KUKA KRL program: MyProgram_289().src

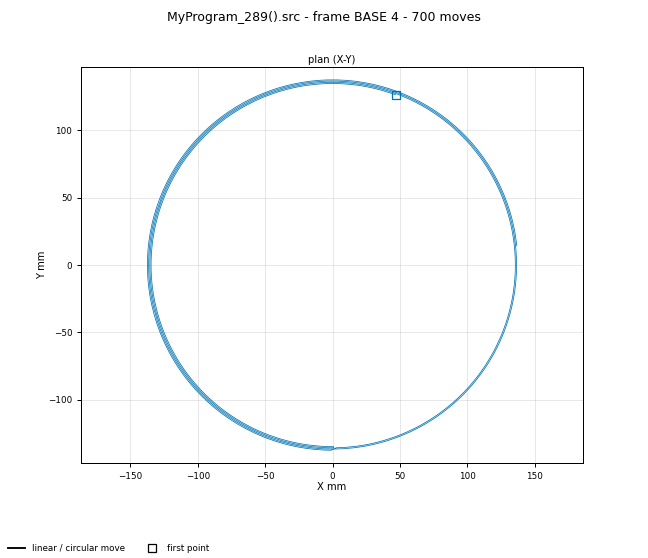
[picture p0: tool path of MyProgram_289().src in frame BASE 4, 700 of 700 moves have a stored position in this frame; points joined in program order, loops and branches not executed]
&ACCESS RVP
&REL 1
&PARAM TEMPLATE = C:\KRC\Roboter\Template\vorgabe
&PARAM EDITMASK = *
DEF MyProgram_289()
; ---- Setting reference (Base) ----
$BASE = BASE_DATA[4]

; --------------------------
; ---- Setting tool (TCP) ----
$TOOL = TOOL_DATA[3]
; --------------------------

$VEL.CP = VEL_APROX_PRINT
Startdeposition()
$VEL.CP = VEL_PRINT
LIN {X 46.739,Y 126.3738,Z 176,A 70.9873,B 7.2165,C 0.098,E1 7.2727,E2 380.9544} C_DIS
LIN {X 43.7934,Y 127.4239,Z 176,A 72.2694,B 7.2165,C 0.0975,E1 7.2693,E2 379.6782} C_DIS
LIN {X 36.8996,Y 129.5888,Z 176,A 75.2053,B 7.2165,C 0.0972,E1 7.2615,E2 376.7596} C_DIS
LIN {X 33.0824,Y 130.6146,Z 176,A 76.9284,B 7.2165,C 0.0952,E1 7.2569,E2 375.0317} C_DIS
LIN {X 29.3241,Y 131.5112,Z 176,A 78.6742,B 7.2166,C 0.0925,E1 7.2521,E2 373.2739} C_DIS
LIN {X 25.3274,Y 132.3373,Z 176,A 80.285,B 7.2166,C 0.0935,E1 7.2477,E2 371.6787} C_DIS
LIN {X 22.0563,Y 132.9217,Z 176,A 81.6963,B 7.2166,C 0.0929,E1 7.2438,E2 370.2679} C_DIS
LIN {X 18.536,Y 133.4592,Z 176,A 83.3203,B 7.2166,C 0.0905,E1 7.2393,E2 368.6313} C_DIS
LIN {X 13.6178,Y 134.0514,Z 176,A 85.4842,B 7.2166,C 0.089,E1 7.2333,E2 366.4611} C_DIS
LIN {X 9.065,Y 134.4361,Z 176,A 87.3794,B 7.2166,C 0.0893,E1 7.228,E2 364.5725} C_DIS
LIN {X 4.9514,Y 134.6487,Z 176,A 88.9717,B 7.2166,C 0.0915,E1 7.2236,E2 363.0001} C_DIS
LIN {X -0.1515,Y 134.74,Z 176,A 91.34,B 7.2166,C 0.0884,E1 7.2169,E2 360.6088} C_DIS
LIN {X -4.7786,Y 134.6554,Z 176,A 93.1801,B 7.2166,C 0.0905,E1 7.2118,E2 358.7852} C_DIS
LIN {X -8.4251,Y 134.4757,Z 176,A 94.6876,B 7.2166,C 0.0914,E1 7.2077,E2 357.2838} C_DIS
LIN {X -12.1995,Y 134.1876,Z 176,A 96.4009,B 7.2166,C 0.0902,E1 7.2029,E2 355.5589} C_DIS
LIN {X -16.1723,Y 133.7653,Z 176,A 97.9295,B 7.2166,C 0.0933,E1 7.1987,E2 354.0517} C_DIS
LIN {X -19.1655,Y 133.3692,Z 176,A 99.271,B 7.2166,C 0.0929,E1 7.1949,E2 352.7039} C_DIS
LIN {X -22.3244,Y 132.8769,Z 176,A 100.6251,B 7.2166,C 0.0936,E1 7.1912,E2 351.3514} C_DIS
LIN {X -25.9494,Y 132.2184,Z 176,A 102.3402,B 7.2166,C 0.0923,E1 7.1865,E2 349.6193} C_DIS
LIN {X -30.1027,Y 131.3334,Z 176,A 104.0357,B 7.2166,C 0.095,E1 7.1819,E2 347.9381} C_DIS
LIN {X -33.5303,Y 130.5009,Z 176,A 105.647,B 7.2166,C 0.0945,E1 7.1775,E2 346.3144} C_DIS
LIN {X -39.6195,Y 128.7825,Z 176,A 108.2833,B 7.2166,C 0.0974,E1 7.1704,E2 343.6864} C_DIS
LIN {X -42.7121,Y 127.79,Z 176,A 110.159,B 7.2166,C 0.0916,E1 7.1653,E2 341.7518} C_DIS
LIN {X -46.9366,Y 126.2998,Z 176,A 111.9973,B 7.2166,C 0.0944,E1 7.1605,E2 339.923} C_DIS
LIN {X -50.7015,Y 124.8361,Z 176,A 113.2648,B 7.2165,C 0.1026,E1 7.1574,E2 338.7113} C_DIS
LIN {X -53.8637,Y 123.5048,Z 176,A 114.743,B 7.2165,C 0.104,E1 7.1536,E2 337.2318} C_DIS
LIN {X -56.9194,Y 122.1266,Z 176,A 116.2037,B 7.2165,C 0.1052,E1 7.1499,E2 335.7679} C_DIS
LIN {X -63.2599,Y 118.9673,Z 176,A 119.0396,B 7.2163,C 0.1116,E1 7.1429,E2 332.9558} C_DIS
LIN {X -65.7728,Y 117.5973,Z 176,A 120.5687,B 7.2163,C 0.109,E1 7.139,E2 331.3901} C_DIS
LIN {X -70.8593,Y 114.6044,Z 176,A 122.972,B 7.2163,C 0.1142,E1 7.1333,E2 329.0017} C_DIS
LIN {X -73.968,Y 112.6226,Z 176,A 124.66,B 7.2163,C 0.115,E1 7.1293,E2 327.3004} C_DIS
LIN {X -78.7898,Y 109.3041,Z 176,A 127.0345,B 7.2163,C 0.1206,E1 7.1239,E2 324.9419} C_DIS
LIN {X -81.5123,Y 107.2894,Z 176,A 128.6056,B 7.2162,C 0.1214,E1 7.1204,E2 323.3563} C_DIS
LIN {X -84.8943,Y 104.6336,Z 176,A 130.4274,B 7.2162,C 0.1248,E1 7.1164,E2 321.5369} C_DIS
LIN {X -87.9949,Y 102.0392,Z 176,A 132.5845,B 7.2162,C 0.1222,E1 7.1117,E2 319.3282} C_DIS
LIN {X -90.9601,Y 99.4054,Z 176,A 133.9926,B 7.2161,C 0.1291,E1 7.1089,E2 317.9555} C_DIS
LIN {X -95.2089,Y 95.344,Z 176,A 136.3018,B 7.2159,C 0.1366,E1 7.1043,E2 315.6716} C_DIS
LIN {X -97.6628,Y 92.8289,Z 176,A 138.2509,B 7.2159,C 0.1338,E1 7.1004,E2 313.6688} C_DIS
LIN {X -99.9947,Y 90.3119,Z 176,A 139.2657,B 7.2158,C 0.1427,E1 7.0986,E2 312.7091} C_DIS
LIN {X -102.1705,Y 87.8423,Z 176,A 141.0418,B 7.2158,C 0.1409,E1 7.0953,E2 310.8887} C_DIS
LIN {X -105.7645,Y 83.4809,Z 176,A 143.5332,B 7.2158,C 0.1452,E1 7.0909,E2 308.3889} C_DIS
LIN {X -108.9535,Y 79.2734,Z 176,A 145.5935,B 7.2156,C 0.1527,E1 7.0875,E2 306.3532} C_DIS
LIN {X -112.011,Y 74.8908,Z 176,A 147.5992,B 7.2154,C 0.1615,E1 7.0844,E2 304.3819} C_DIS
LIN {X -113.5489,Y 72.538,Z 176,A 149.4424,B 7.2155,C 0.1562,E1 7.0815,E2 302.4612} C_DIS
LIN {X -115.46,Y 69.4557,Z 176,A 150.6583,B 7.2153,C 0.1642,E1 7.0798,E2 301.2866} C_DIS
LIN {X -117.0516,Y 66.7384,Z 176,A 152.5358,B 7.2154,C 0.1607,E1 7.0771,E2 299.3447} C_DIS
LIN {X -119.1423,Y 62.9266,Z 176,A 153.6832,B 7.2151,C 0.1743,E1 7.0757,E2 298.2845} C_DIS
LIN {X -120.2429,Y 60.7975,Z 176,A 154.9377,B 7.2151,C 0.1739,E1 7.0741,E2 297.0024} C_DIS
LIN {X -121.7624,Y 57.6944,Z 176,A 156.459,B 7.2151,C 0.1771,E1 7.0722,E2 295.4761} C_DIS
LIN {X -123.8033,Y 53.1733,Z 176,A 158.5577,B 7.2149,C 0.1828,E1 7.0699,E2 293.3808} C_DIS
LIN {X -125.0493,Y 50.1725,Z 176,A 160.0003,B 7.2149,C 0.1857,E1 7.0683,E2 291.9321} C_DIS
LIN {X -127.412,Y 43.8276,Z 176,A 162.9337,B 7.2146,C 0.1929,E1 7.0655,E2 288.9949} C_DIS
LIN {X -128.6112,Y 40.1791,Z 176,A 164.7288,B 7.2146,C 0.1954,E1 7.064,E2 287.1816} C_DIS
LIN {X -129.7986,Y 36.1515,Z 176,A 166.3975,B 7.2144,C 0.2018,E1 7.0627,E2 285.5288} C_DIS
LIN {X -130.7393,Y 32.5908,Z 176,A 167.9676,B 7.2143,C 0.2061,E1 7.0616,E2 283.9597} C_DIS
LIN {X -131.4143,Y 29.7485,Z 176,A 169.2369,B 7.2142,C 0.2092,E1 7.0608,E2 282.6882} C_DIS
LIN {X -132.1055,Y 26.5122,Z 176,A 170.6847,B 7.2141,C 0.2127,E1 7.06,E2 281.2367} C_DIS
LIN {X -132.7822,Y 22.8924,Z 176,A 172.4282,B 7.2141,C 0.215,E1 7.0591,E2 279.473} C_DIS
LIN {X -133.3823,Y 19.0741,Z 176,A 173.9886,B 7.2138,C 0.2207,E1 7.0585,E2 277.9242} C_DIS
LIN {X -133.8523,Y 15.4428,Z 176,A 175.6627,B 7.2138,C 0.2237,E1 7.0579,E2 276.2371} C_DIS
LIN {X -134.2767,Y 11.1572,Z 176,A 177.4463,B 7.2136,C 0.2295,E1 7.0575,E2 274.461} C_DIS
LIN {X -134.5431,Y 7.2873,Z 176,A 179.2247,B 7.2135,C 0.2327,E1 7.0572,E2 272.6683} C_DIS
LIN {X -134.7031,Y 3.1775,Z 176,A -178.9548,B 7.2133,C 0.2368,E1 7.057,E2 270.8405} C_DIS
LIN {X -134.7368,Y -0.9717,Z 176,A -177.1983,B 7.2132,C 0.242,E1 7.057,E2 269.0864} C_DIS
LIN {X -134.6421,Y -5.1206,Z 176,A -175.4593,B 7.213,C 0.2474,E1 7.0572,E2 267.352} C_DIS
LIN {X -134.429,Y -9.1625,Z 176,A -173.6351,B 7.2129,C 0.251,E1 7.0575,E2 265.5166} C_DIS
LIN {X -134.1144,Y -12.9613,Z 176,A -172.077,B 7.2127,C 0.2564,E1 7.0579,E2 263.9675} C_DIS
LIN {X -133.7153,Y -16.5917,Z 176,A -170.4743,B 7.2125,C 0.2602,E1 7.0584,E2 262.36} C_DIS
LIN {X -133.1806,Y -20.4353,Z 176,A -168.761,B 7.2124,C 0.2641,E1 7.0591,E2 260.6401} C_DIS
LIN {X -132.5589,Y -24.1444,Z 176,A -167.1691,B 7.2122,C 0.2687,E1 7.0599,E2 259.0503} C_DIS
LIN {X -131.7289,Y -28.322,Z 176,A -165.3319,B 7.212,C 0.2735,E1 7.0609,E2 257.2112} C_DIS
LIN {X -130.0027,Y -35.4179,Z 176,A -161.457,B 7.212,C 0.2724,E1 7.0637,E2 253.2431} C_DIS
LIN {X -128.5121,Y -40.4909,Z 176,A -159.9882,B 7.2115,C 0.2884,E1 7.0648,E2 251.8727} C_DIS
LIN {X -127.1443,Y -44.5999,Z 176,A -157.774,B 7.2115,C 0.2886,E1 7.0668,E2 249.6135} C_DIS
LIN {X -125.5592,Y -48.882,Z 176,A -155.9827,B 7.2112,C 0.2957,E1 7.0686,E2 247.8421} C_DIS
LIN {X -124.2324,Y -52.1626,Z 176,A -154.4732,B 7.211,C 0.2996,E1 7.0702,E2 246.333} C_DIS
LIN {X -122.9434,Y -55.1316,Z 176,A -153.0961,B 7.2109,C 0.3031,E1 7.0717,E2 244.9566} C_DIS
LIN {X -121.2485,Y -58.7688,Z 176,A -151.3637,B 7.2107,C 0.3072,E1 7.0738,E2 243.2219} C_DIS
LIN {X -120.0628,Y -61.1512,Z 176,A -149.7902,B 7.2108,C 0.3043,E1 7.0759,E2 241.5939} C_DIS
LIN {X -118.2615,Y -64.5696,Z 176,A -148.0643,B 7.2107,C 0.3073,E1 7.0782,E2 239.8586} C_DIS
LIN {X -116.2697,Y -68.0917,Z 176,A -147.0058,B 7.2101,C 0.3201,E1 7.0796,E2 238.8836} C_DIS
LIN {X -114.7894,Y -70.5584,Z 176,A -145.4501,B 7.2101,C 0.3188,E1 7.0819,E2 237.2872} C_DIS
LIN {X -112.3758,Y -74.3429,Z 176,A -143.133,B 7.2102,C 0.3179,E1 7.0855,E2 234.9198} C_DIS
LIN {X -110.1367,Y -77.6209,Z 176,A -141.8141,B 7.2098,C 0.3267,E1 7.0875,E2 233.6479} C_DIS
LIN {X -108.2709,Y -80.2035,Z 176,A -139.8806,B 7.2101,C 0.3221,E1 7.0909,E2 231.6424} C_DIS
LIN {X -105.3441,Y -84.0103,Z 176,A -138.3443,B 7.2095,C 0.3333,E1 7.0934,E2 230.1703} C_DIS
LIN {X -102.7193,Y -87.2,Z 176,A -136.5236,B 7.2095,C 0.3362,E1 7.0967,E2 228.3423} C_DIS
LIN {X -99.0727,Y -91.322,Z 176,A -134.4345,B 7.209,C 0.3444,E1 7.1005,E2 226.2854} C_DIS
LIN {X -97.1061,Y -93.4113,Z 176,A -132.8728,B 7.2091,C 0.3423,E1 7.1036,E2 224.6813} C_DIS
LIN {X -93.9427,Y -96.5917,Z 176,A -130.9489,B 7.209,C 0.3457,E1 7.1074,E2 222.7558} C_DIS
LIN {X -90.755,Y -99.5926,Z 176,A -129.0641,B 7.2088,C 0.3489,E1 7.1113,E2 220.8685} C_DIS
LIN {X -87.4295,Y -102.5242,Z 176,A -127.1743,B 7.2086,C 0.3522,E1 7.1153,E2 218.9786} C_DIS
LIN {X -83.2923,Y -105.9126,Z 176,A -125.0607,B 7.2083,C 0.3584,E1 7.1199,E2 216.8855} C_DIS
LIN {X -80.0894,Y -108.3546,Z 176,A -122.7965,B 7.2086,C 0.3535,E1 7.1251,E2 214.5521} C_DIS
LIN {X -76.7889,Y -110.7185,Z 176,A -121.6345,B 7.2081,C 0.3641,E1 7.1276,E2 213.4614} C_DIS
LIN {X -73.9442,Y -112.6382,Z 176,A -119.9283,B 7.2081,C 0.3628,E1 7.1316,E2 211.7243} C_DIS
LIN {X -70.1568,Y -115.0358,Z 176,A -117.9951,B 7.2081,C 0.3651,E1 7.1362,E2 209.7879} C_DIS
LIN {X -66.356,Y -117.2694,Z 176,A -116.0672,B 7.2079,C 0.3669,E1 7.1409,E2 207.8532} C_DIS
LIN {X -62.4442,Y -119.3956,Z 176,A -114.285,B 7.2077,C 0.3708,E1 7.1452,E2 206.0849} C_DIS
LIN {X -59.2266,Y -121.0245,Z 176,A -112.754,B 7.2077,C 0.3727,E1 7.1491,E2 204.5543} C_DIS
LIN {X -55.9568,Y -122.5717,Z 176,A -111.1959,B 7.2076,C 0.3741,E1 7.153,E2 202.9936} C_DIS
LIN {X -51.5409,Y -124.492,Z 176,A -109.084,B 7.2075,C 0.3753,E1 7.1585,E2 200.8733} C_DIS
LIN {X -46.8002,Y -126.3509,Z 176,A -106.8561,B 7.2075,C 0.3763,E1 7.1643,E2 198.6373} C_DIS
LIN {X -40.0759,Y -128.6423,Z 176,A -103.9389,B 7.2072,C 0.3803,E1 7.172,E2 195.7328} C_DIS
LIN {X -37.4879,Y -129.4195,Z 176,A -102.7989,B 7.2072,C 0.3812,E1 7.175,E2 194.5936} C_DIS
LIN {X -34.6618,Y -130.2043,Z 176,A -101.5236,B 7.2072,C 0.3816,E1 7.1785,E2 193.3145} C_DIS
LIN {X -31.4986,Y -131.0055,Z 176,A -100.1131,B 7.2072,C 0.382,E1 7.1823,E2 191.9007} C_DIS
LIN {X -28.3558,Y -131.7216,Z 176,A -98.766,B 7.2071,C 0.3831,E1 7.186,E2 190.5562} C_DIS
LIN {X -25.1394,Y -132.3732,Z 176,A -97.3637,B 7.2071,C 0.3836,E1 7.1898,E2 189.1526} C_DIS
LIN {X -22.007,Y -132.9299,Z 176,A -95.9846,B 7.2071,C 0.3836,E1 7.1936,E2 187.7698} C_DIS
LIN {X -18.2836,Y -133.4951,Z 176,A -93.8301,B 7.2075,C 0.3755,E1 7.1998,E2 185.5446} C_DIS
LIN {X -13.7352,Y -134.0391,Z 176,A -92.4659,B 7.207,C 0.3851,E1 7.2034,E2 184.2538} C_DIS
LIN {X -10.8566,Y -134.3021,Z 176,A -91.1132,B 7.207,C 0.3833,E1 7.2072,E2 182.885} C_DIS
LIN {X -6.8342,Y -134.5659,Z 176,A -89.1612,B 7.2073,C 0.3795,E1 7.2127,E2 180.902} C_DIS
LIN {X -3.396,Y -134.697,Z 176,A -87.6016,B 7.2073,C 0.3779,E1 7.2171,E2 179.3295} C_DIS
LIN {X 0.5077,Y -134.7387,Z 176,A -86.3072,B 7.2071,C 0.3836,E1 7.2206,E2 178.0808} C_DIS
LIN {X 0.5077,Y -134.7387,Z 176,A -86.3072,B 7.2071,C 0.3836,E1 7.2206,E2 178.0808} C_DIS
Enddeposition()
LIN {X 0.996,Y -135.641,Z 176,A -86.1239,B 7.1241,C 0.3885,E1 7.1383,E2 177.9572} C_DIS
Startdeposition()
$VEL.CP = VEL_PRINT
LIN {X -4.7077,Y -135.5642,Z 176,A -89.0853,B 7.1236,C 0.3974,E1 7.1299,E2 180.9899} C_DIS
LIN {X -9.5873,Y -135.3061,Z 176,A -91.2415,B 7.1236,C 0.3987,E1 7.1238,E2 183.1586} C_DIS
LIN {X -13.0181,Y -135.0188,Z 176,A -93.0667,B 7.1232,C 0.4042,E1 7.1186,E2 185.0311} C_DIS
LIN {X -16.8806,Y -134.5909,Z 176,A -94.558,B 7.1234,C 0.4015,E1 7.1145,E2 186.5041} C_DIS
LIN {X -22.3201,Y -133.7959,Z 176,A -96.6569,B 7.1236,C 0.3974,E1 7.1088,E2 188.5757} C_DIS
LIN {X -26.2786,Y -133.0773,Z 176,A -98.4709,B 7.1236,C 0.3984,E1 7.1038,E2 190.4048} C_DIS
LIN {X -30.3133,Y -132.2143,Z 176,A -100.0712,B 7.1236,C 0.3954,E1 7.0995,E2 191.9875} C_DIS
LIN {X -33.4857,Y -131.4466,Z 176,A -101.4995,B 7.1236,C 0.3954,E1 7.0956,E2 193.4224} C_DIS
LIN {X -36.965,Y -130.5116,Z 176,A -103.0564,B 7.1237,C 0.3949,E1 7.0914,E2 194.9841} C_DIS
LIN {X -43.7768,Y -128.3882,Z 176,A -105.9689,B 7.1239,C 0.3911,E1 7.0837,E2 197.8845} C_DIS
LIN {X -47.6211,Y -127.0106,Z 176,A -107.8293,B 7.1239,C 0.3916,E1 7.0787,E2 199.7621} C_DIS
LIN {X -51.2699,Y -125.5835,Z 176,A -109.6042,B 7.1239,C 0.3917,E1 7.0741,E2 201.5524} C_DIS
LIN {X -54.6493,Y -124.1513,Z 176,A -110.9764,B 7.1241,C 0.3876,E1 7.0706,E2 202.9023} C_DIS
LIN {X -57.1447,Y -123.0202,Z 176,A -112.1786,B 7.1241,C 0.3869,E1 7.0676,E2 204.1103} C_DIS
LIN {X -60.2043,Y -121.5521,Z 176,A -113.6365,B 7.1242,C 0.3856,E1 7.0639,E2 205.5713} C_DIS
LIN {X -63.7521,Y -119.7318,Z 176,A -115.3454,B 7.1243,C 0.3839,E1 7.0597,E2 207.2833} C_DIS
LIN {X -67.5396,Y -117.6373,Z 176,A -117.2786,B 7.1243,C 0.383,E1 7.0549,E2 209.2297} C_DIS
LIN {X -71.4568,Y -115.2995,Z 176,A -119.2047,B 7.1245,C 0.3803,E1 7.0503,E2 211.1557} C_DIS
LIN {X -75.2415,Y -112.8659,Z 176,A -121.1047,B 7.1247,C 0.3775,E1 7.0459,E2 213.0554} C_DIS
LIN {X -80.6564,Y -109.0628,Z 176,A -123.9768,B 7.1248,C 0.3741,E1 7.0393,E2 215.9369} C_DIS
LIN {X -84.2255,Y -106.3303,Z 176,A -125.9951,B 7.1249,C 0.3725,E1 7.0349,E2 217.9698} C_DIS
LIN {X -87.0011,Y -104.0714,Z 176,A -127.4206,B 7.1251,C 0.3687,E1 7.0318,E2 219.3843} C_DIS
LIN {X -90.5428,Y -101.0048,Z 176,A -129.3934,B 7.1253,C 0.3651,E1 7.0277,E2 221.356} C_DIS
LIN {X -93.9342,Y -97.8593,Z 176,A -131.3841,B 7.1255,C 0.3618,E1 7.0236,E2 223.3508} C_DIS
LIN {X -97.1434,Y -94.6747,Z 176,A -133.3331,B 7.1256,C 0.3586,E1 7.0198,E2 225.3042} C_DIS
LIN {X -100.7337,Y -90.8447,Z 176,A -135.4229,B 7.1259,C 0.3524,E1 7.0159,E2 227.3774} C_DIS
LIN {X -102.6613,Y -88.6604,Z 176,A -136.8314,B 7.1259,C 0.3522,E1 7.0132,E2 228.8076} C_DIS
LIN {X -105.5562,Y -85.1931,Z 176,A -138.734,B 7.1262,C 0.348,E1 7.0099,E2 230.7089} C_DIS
LIN {X -110.1768,Y -79.1273,Z 176,A -141.7148,B 7.1266,C 0.3377,E1 7.0049,E2 233.6586} C_DIS
LIN {X -113.3344,Y -74.5338,Z 176,A -144.1448,B 7.1269,C 0.3332,E1 7.0011,E2 236.0971} C_DIS
LIN {X -114.9573,Y -72.0066,Z 176,A -145.7504,B 7.1268,C 0.3345,E1 6.9986,E2 237.744} C_DIS
LIN {X -117.317,Y -68.0936,Z 176,A -148.2444,B 7.1267,C 0.3369,E1 6.995,E2 240.3066} C_DIS
LIN {X -119.8043,Y -63.614,Z 176,A -149.6976,B 7.1273,C 0.3226,E1 6.9932,E2 241.671} C_DIS
LIN {X -121.1064,Y -61.0976,Z 176,A -151.0675,B 7.1273,C 0.3218,E1 6.9914,E2 243.0616} C_DIS
LIN {X -123.2128,Y -56.7282,Z 176,A -153.0883,B 7.1276,C 0.3162,E1 6.989,E2 245.0778} C_DIS
LIN {X -124.5702,Y -53.6818,Z 176,A -154.5239,B 7.1278,C 0.3129,E1 6.9874,E2 246.5159} C_DIS
LIN {X -125.973,Y -50.3035,Z 176,A -156.101,B 7.1279,C 0.3092,E1 6.9857,E2 248.096} C_DIS
LIN {X -127.2111,Y -47.0857,Z 176,A -157.6421,B 7.1281,C 0.3064,E1 6.9842,E2 249.6467} C_DIS
LIN {X -128.4332,Y -43.6467,Z 176,A -159.1463,B 7.1282,C 0.3018,E1 6.9828,E2 251.1454} C_DIS
LIN {X -129.8934,Y -39.0844,Z 176,A -161.797,B 7.1282,C 0.304,E1 6.9806,E2 253.8717} C_DIS
LIN {X -131.1515,Y -34.6251,Z 176,A -163.5893,B 7.1285,C 0.2966,E1 6.9793,E2 255.6424} C_DIS
LIN {X -132.063,Y -30.9751,Z 176,A -164.8088,B 7.1288,C 0.2876,E1 6.9785,E2 256.8155} C_DIS
LIN {X -132.9914,Y -26.7009,Z 176,A -166.6352,B 7.129,C 0.2822,E1 6.9775,E2 258.6379} C_DIS
LIN {X -133.5606,Y -23.6881,Z 176,A -168.0202,B 7.1291,C 0.2797,E1 6.9768,E2 260.0329} C_DIS
LIN {X -134.1555,Y -20.0583,Z 176,A -169.789,B 7.1292,C 0.2779,E1 6.976,E2 261.827} C_DIS
LIN {X -134.6974,Y -16.0048,Z 176,A -171.411,B 7.1295,C 0.2717,E1 6.9754,E2 263.4348} C_DIS
LIN {X -135.117,Y -11.9696,Z 176,A -173.227,B 7.1295,C 0.2681,E1 6.9749,E2 265.262} C_DIS
LIN {X -135.4001,Y -8.1499,Z 176,A -174.7919,B 7.1298,C 0.2628,E1 6.9746,E2 266.8191} C_DIS
LIN {X -135.5792,Y -4.2544,Z 176,A -176.5543,B 7.1299,C 0.2595,E1 6.9745,E2 268.5943} C_DIS
LIN {X -135.6467,Y -0.306,Z 176,A -178.188,B 7.1301,C 0.2543,E1 6.9745,E2 270.2224} C_DIS
LIN {X -135.5959,Y 3.6532,Z 176,A -179.9351,B 7.1302,C 0.2504,E1 6.9745,E2 271.9772} C_DIS
LIN {X -135.4109,Y 7.9751,Z 176,A 178.1962,B 7.1304,C 0.2456,E1 6.9748,E2 273.8494} C_DIS
LIN {X -135.1544,Y 11.5263,Z 176,A 176.6976,B 7.1305,C 0.2412,E1 6.9751,E2 275.3459} C_DIS
LIN {X -134.7366,Y 15.6763,Z 176,A 174.8477,B 7.1307,C 0.2373,E1 6.9756,E2 277.205} C_DIS
LIN {X -134.27,Y 19.264,Z 176,A 173.3565,B 7.1308,C 0.2325,E1 6.9762,E2 278.6904} C_DIS
LIN {X -133.7599,Y 22.5356,Z 176,A 171.8778,B 7.1309,C 0.2294,E1 6.9769,E2 280.1776} C_DIS
LIN {X -132.9543,Y 26.8828,Z 176,A 170.0024,B 7.1311,C 0.2243,E1 6.9779,E2 282.0523} C_DIS
LIN {X -132.2009,Y 30.3717,Z 176,A 168.4755,B 7.1312,C 0.2203,E1 6.9788,E2 283.5801} C_DIS
LIN {X -131.3092,Y 34.0272,Z 176,A 166.6861,B 7.1312,C 0.2182,E1 6.98,E2 285.3924} C_DIS
LIN {X -130.1443,Y 38.2357,Z 176,A 164.9617,B 7.1315,C 0.2117,E1 6.9813,E2 287.1004} C_DIS
LIN {X -128.9768,Y 42.0127,Z 176,A 162.8066,B 7.1315,C 0.2129,E1 6.9832,E2 289.3128} C_DIS
LIN {X -127.6927,Y 45.7614,Z 176,A 161.1611,B 7.1315,C 0.208,E1 6.9848,E2 290.9532} C_DIS
LIN {X -126.3735,Y 49.2871,Z 176,A 159.9412,B 7.1318,C 0.1993,E1 6.9859,E2 292.1268} C_DIS
LIN {X -125.0343,Y 52.5927,Z 176,A 158.3786,B 7.1319,C 0.196,E1 6.9876,E2 293.6948} C_DIS
LIN {X -123.749,Y 55.5487,Z 176,A 156.9618,B 7.132,C 0.193,E1 6.9892,E2 295.1171} C_DIS
LIN {X -121.9613,Y 59.3748,Z 176,A 155.0967,B 7.132,C 0.1894,E1 6.9915,E2 296.9904} C_DIS
LIN {X -120.2137,Y 62.8344,Z 176,A 152.9644,B 7.132,C 0.1912,E1 6.9943,E2 299.1805} C_DIS
LIN {X -117.9396,Y 67.0095,Z 176,A 151.4736,B 7.1323,C 0.1799,E1 6.9962,E2 300.6073} C_DIS
LIN {X -114.947,Y 72.0231,Z 176,A 149.1216,B 7.1325,C 0.1724,E1 6.9996,E2 302.9432} C_DIS
LIN {X -113.2159,Y 74.7139,Z 176,A 147.4934,B 7.1325,C 0.1725,E1 7.0021,E2 304.6036} C_DIS
LIN {X -110.5111,Y 78.6598,Z 176,A 145.412,B 7.1326,C 0.1685,E1 7.0055,E2 306.6903} C_DIS
LIN {X -107.3939,Y 82.8645,Z 176,A 143.3778,B 7.1328,C 0.1612,E1 7.0088,E2 308.7012} C_DIS
LIN {X -105.7022,Y 85.0121,Z 176,A 142.0358,B 7.1328,C 0.1609,E1 7.0112,E2 310.0647} C_DIS
LIN {X -102.2429,Y 89.1424,Z 176,A 139.7364,B 7.1328,C 0.1562,E1 7.0154,E2 312.3649} C_DIS
LIN {X -98.349,Y 93.4217,Z 176,A 137.3126,B 7.133,C 0.1508,E1 7.02,E2 314.784} C_DIS
LIN {X -95.5885,Y 96.2435,Z 176,A 135.0858,B 7.133,C 0.1545,E1 7.0245,E2 317.0763} C_DIS
LIN {X -92.2942,Y 99.4072,Z 176,A 133.0505,B 7.133,C 0.1521,E1 7.0287,E2 319.1225} C_DIS
LIN {X -88.5973,Y 102.7157,Z 176,A 131.6203,B 7.1332,C 0.1396,E1 7.0315,E2 320.4713} C_DIS
LIN {X -85.7718,Y 105.0866,Z 176,A 129.8866,B 7.1332,C 0.139,E1 7.0353,E2 322.2247} C_DIS
LIN {X -82.7111,Y 107.5128,Z 176,A 128.1632,B 7.1332,C 0.137,E1 7.0391,E2 323.9556} C_DIS
LIN {X -78.4225,Y 110.6788,Z 176,A 125.9224,B 7.1334,C 0.1331,E1 7.0441,E2 326.1931} C_DIS
LIN {X -75.3263,Y 112.8093,Z 176,A 124.3183,B 7.1334,C 0.1307,E1 7.0479,E2 327.7979} C_DIS
LIN {X -71.4969,Y 115.2745,Z 176,A 121.5698,B 7.1333,C 0.1387,E1 7.0546,E2 330.643} C_DIS
LIN {X -65.9584,Y 118.5308,Z 176,A 119.6722,B 7.1335,C 0.124,E1 7.059,E2 332.4413} C_DIS
LIN {X -58.2367,Y 122.5071,Z 176,A 116.0304,B 7.1336,C 0.1189,E1 7.068,E2 336.0772} C_DIS
LIN {X -55.0069,Y 123.9913,Z 176,A 114.4758,B 7.1336,C 0.1178,E1 7.072,E2 337.637} C_DIS
LIN {X -51.4984,Y 125.4913,Z 176,A 111.9759,B 7.1335,C 0.1282,E1 7.0788,E2 340.2415} C_DIS
LIN {X -45.5058,Y 127.7848,Z 176,A 110.1969,B 7.1337,C 0.1127,E1 7.0831,E2 341.9077} C_DIS
LIN {X -42.6383,Y 128.7691,Z 176,A 108.8279,B 7.1337,C 0.1127,E1 7.0868,E2 343.2864} C_DIS
LIN {X -39.2995,Y 129.8276,Z 176,A 106.9759,B 7.1337,C 0.1168,E1 7.0918,E2 345.182} C_DIS
LIN {X -35.5706,Y 130.8993,Z 176,A 105.8086,B 7.1337,C 0.1089,E1 7.0948,E2 346.2919} C_DIS
LIN {X -32.1245,Y 131.7863,Z 176,A 104.1734,B 7.1337,C 0.1097,E1 7.0993,E2 347.942} C_DIS
LIN {X -28.5733,Y 132.6012,Z 176,A 102.6646,B 7.1337,C 0.1083,E1 7.1034,E2 349.4462} C_DIS
LIN {X -24.9362,Y 133.3342,Z 176,A 101.138,B 7.1338,C 0.1069,E1 7.1075,E2 350.967} C_DIS
LIN {X -21.8816,Y 133.869,Z 176,A 99.7491,B 7.1338,C 0.1074,E1 7.1114,E2 352.3647} C_DIS
LIN {X -17.8333,Y 134.4677,Z 176,A 98.0158,B 7.1338,C 0.1068,E1 7.1162,E2 354.0976} C_DIS
LIN {X -14.0847,Y 134.9124,Z 176,A 96.3394,B 7.1338,C 0.1075,E1 7.1209,E2 355.7829} C_DIS
LIN {X -9.9702,Y 135.2781,Z 176,A 94.6732,B 7.1338,C 0.106,E1 7.1255,E2 357.4388} C_DIS
LIN {X -6.0142,Y 135.5136,Z 176,A 92.8868,B 7.1338,C 0.1074,E1 7.1305,E2 359.2379} C_DIS
LIN {X -1.7426,Y 135.6343,Z 176,A 91.0375,B 7.1338,C 0.108,E1 7.1357,E2 361.0916} C_DIS
LIN {X 3.4099,Y 135.6027,Z 176,A 89.0337,B 7.1338,C 0.1055,E1 7.1412,E2 363.0737} C_DIS
LIN {X 6.5509,Y 135.487,Z 176,A 87.6793,B 7.1338,C 0.106,E1 7.145,E2 364.4308} C_DIS
LIN {X 10.1232,Y 135.267,Z 176,A 86.132,B 7.1338,C 0.1069,E1 7.1493,E2 365.9817} C_DIS
LIN {X 14.2563,Y 134.8939,Z 176,A 84.4263,B 7.1338,C 0.1067,E1 7.154,E2 367.6812} C_DIS
LIN {X 18.3399,Y 134.4013,Z 176,A 82.5974,B 7.1338,C 0.1087,E1 7.1591,E2 369.5205} C_DIS
LIN {X 22.296,Y 133.7999,Z 176,A 81.0367,B 7.1338,C 0.1075,E1 7.1634,E2 371.0651} C_DIS
LIN {X 25.7585,Y 133.177,Z 176,A 79.565,B 7.1338,C 0.1081,E1 7.1674,E2 372.5347} C_DIS
LIN {X 28.7296,Y 132.5674,Z 176,A 78.3064,B 7.1338,C 0.1085,E1 7.1709,E2 373.7902} C_DIS
LIN {X 31.9423,Y 131.8302,Z 176,A 76.8821,B 7.1338,C 0.1099,E1 7.1747,E2 375.218} C_DIS
LIN {X 35.7578,Y 130.8492,Z 176,A 74.5988,B 7.1336,C 0.1209,E1 7.1811,E2 377.5752} C_DIS
LIN {X 40.665,Y 129.4073,Z 176,A 73.1781,B 7.1337,C 0.111,E1 7.1847,E2 378.9069} C_DIS
LIN {X 45.3873,Y 127.8276,Z 176,A 71.001,B 7.1337,C 0.1141,E1 7.1904,E2 381.0925} C_DIS
LIN {X 48.392,Y 126.7214,Z 176,A 69.4815,B 7.1337,C 0.1182,E1 7.1945,E2 382.6319} C_DIS
LIN {X 52.4009,Y 125.1144,Z 176,A 67.8358,B 7.1337,C 0.1173,E1 7.1986,E2 384.2559} C_DIS
LIN {X 55.5295,Y 123.7576,Z 176,A 66.4224,B 7.1337,C 0.1185,E1 7.2023,E2 385.666} C_DIS
LIN {X 58.659,Y 122.3054,Z 176,A 64.9734,B 7.1336,C 0.1202,E1 7.2059,E2 387.1138} C_DIS
LIN {X 61.9204,Y 120.6875,Z 176,A 63.4073,B 7.1336,C 0.1226,E1 7.2098,E2 388.6834} C_DIS
LIN {X 66.0072,Y 118.5038,Z 176,A 61.4124,B 7.1335,C 0.126,E1 7.2147,E2 390.6829} C_DIS
LIN {X 69.864,Y 116.2719,Z 176,A 59.5271,B 7.1335,C 0.1288,E1 7.2193,E2 392.5686} C_DIS
LIN {X 73.7625,Y 113.838,Z 176,A 57.4366,B 7.1333,C 0.1342,E1 7.2242,E2 394.6773} C_DIS
LIN {X 76.5449,Y 111.9863,Z 176,A 56.522,B 7.1335,C 0.1282,E1 7.2262,E2 395.5319} C_DIS
LIN {X 78.968,Y 110.2907,Z 176,A 55.0286,B 7.1333,C 0.1344,E1 7.2297,E2 397.055} C_DIS
LIN {X 82.6447,Y 107.5636,Z 176,A 53.1043,B 7.1333,C 0.1375,E1 7.234,E2 398.9785} C_DIS
LIN {X 86.0394,Y 104.8678,Z 176,A 51.2855,B 7.1333,C 0.1406,E1 7.2379,E2 400.7961} C_DIS
LIN {X 89.5419,Y 101.894,Z 176,A 49.3471,B 7.1331,C 0.1442,E1 7.242,E2 402.7346} C_DIS
LIN {X 94.0074,Y 97.789,Z 176,A 46.9457,B 7.1331,C 0.1464,E1 7.2469,E2 405.1172} C_DIS
LIN {X 96.9655,Y 94.8562,Z 176,A 44.8539,B 7.1329,C 0.1558,E1 7.2511,E2 407.2497} C_DIS
LIN {X 99.4961,Y 92.1988,Z 176,A 43.8957,B 7.1331,C 0.1487,E1 7.2528,E2 408.1365} C_DIS
LIN {X 102.8361,Y 88.4575,Z 176,A 41.533,B 7.1329,C 0.1575,E1 7.2572,E2 410.5296} C_DIS
LIN {X 107.0011,Y 83.3719,Z 176,A 39.0545,B 7.1329,C 0.1585,E1 7.2615,E2 412.9728} C_DIS
LIN {X 109.9809,Y 79.3993,Z 176,A 36.7545,B 7.1327,C 0.1669,E1 7.2654,E2 415.2985} C_DIS
LIN {X 112.3078,Y 76.0719,Z 176,A 35.0364,B 7.1326,C 0.1709,E1 7.2681,E2 417.0177} C_DIS
LIN {X 114.769,Y 72.3054,Z 176,A 33.189,B 7.1325,C 0.1746,E1 7.2709,E2 418.8594} C_DIS
LIN {X 116.9891,Y 68.6551,Z 176,A 31.4003,B 7.1324,C 0.1787,E1 7.2734,E2 420.647} C_DIS
LIN {X 119.1728,Y 64.7909,Z 176,A 29.5432,B 7.1323,C 0.1831,E1 7.2759,E2 422.5029} C_DIS
LIN {X 121.0138,Y 61.2794,Z 176,A 28.0036,B 7.1323,C 0.1849,E1 7.2779,E2 424.0268} C_DIS
LIN {X 122.446,Y 58.3646,Z 176,A 26.6283,B 7.1321,C 0.1885,E1 7.2796,E2 425.4033} C_DIS
LIN {X 124.0324,Y 54.9152,Z 176,A 24.9355,B 7.132,C 0.1943,E1 7.2815,E2 427.108} C_DIS
LIN {X 125.9016,Y 50.4808,Z 176,A 22.848,B 7.1318,C 0.2007,E1 7.2838,E2 429.2033} C_DIS
LIN {X 127.8599,Y 45.2975,Z 176,A 20.7871,B 7.1318,C 0.2019,E1 7.2857,E2 431.2315} C_DIS
LIN {X 128.9019,Y 42.2396,Z 176,A 19.3451,B 7.1316,C 0.207,E1 7.287,E2 432.6839} C_DIS
LIN {X 130.1492,Y 38.2188,Z 176,A 17.7161,B 7.1316,C 0.2091,E1 7.2883,E2 434.2956} C_DIS
LIN {X 131.0707,Y 34.928,Z 176,A 16.2916,B 7.1314,C 0.2128,E1 7.2894,E2 435.7188} C_DIS
LIN {X 131.8984,Y 31.6596,Z 176,A 14.8757,B 7.1314,C 0.2166,E1 7.2903,E2 437.1347} C_DIS
LIN {X 132.6614,Y 28.2944,Z 176,A 13.4527,B 7.1312,C 0.22,E1 7.2912,E2 438.5545} C_DIS
LIN {X 133.4327,Y 24.4028,Z 176,A 11.7073,B 7.131,C 0.226,E1 7.2921,E2 440.3098} C_DIS
LIN {X 134.134,Y 20.1968,Z 176,A 10.0006,B 7.131,C 0.2294,E1 7.2928,E2 442.0062} C_DIS
LIN {X 134.6848,Y 16.1111,Z 176,A 8.3269,B 7.1308,C 0.2331,E1 7.2934,E2 443.6728} C_DIS
LIN {X 135.0735,Y 12.449,Z 176,A 6.6976,B 7.1306,C 0.2389,E1 7.2939,E2 445.3125} C_DIS
LIN {X 135.4138,Y 7.9278,Z 176,A 4.9177,B 7.1306,C 0.2419,E1 7.2942,E2 447.0772} C_DIS
LIN {X 135.5861,Y 4.0082,Z 176,A 3.1359,B 7.1303,C 0.249,E1 7.2944,E2 448.8757} C_DIS
LIN {X 135.6457,Y 0.456,Z 176,A 1.8125,B 7.1303,C 0.25,E1 7.2944,E2 450.1785} C_DIS
LIN {X 135.593,Y -3.7595,Z 176,A -0.5402,B 7.1297,C 0.2657,E1 7.2942,E2 452.6033} C_DIS
LIN {X 135.3526,Y -8.8953,Z 176,A -1.9947,B 7.1299,C 0.2587,E1 7.294,E2 453.971} C_DIS
LIN {X 135.0885,Y -12.2926,Z 176,A -3.3755,B 7.1299,C 0.2617,E1 7.2937,E2 455.346} C_DIS
LIN {X 134.56,Y -17.1289,Z 176,A -5.5523,B 7.1295,C 0.2699,E1 7.293,E2 457.5396} C_DIS
LIN {X 134.0147,Y -20.9674,Z 176,A -7.1078,B 7.1295,C 0.273,E1 7.2924,E2 459.0864} C_DIS
LIN {X 133.2434,Y -25.4111,Z 176,A -8.9627,B 7.1292,C 0.2775,E1 7.2914,E2 460.9368} C_DIS
LIN {X 132.532,Y -28.8936,Z 176,A -10.4262,B 7.1291,C 0.281,E1 7.2906,E2 462.397} C_DIS
LIN {X 130.7885,Y -35.975,Z 176,A -13.3191,B 7.1289,C 0.2862,E1 7.2886,E2 465.2694} C_DIS
LIN {X 129.5654,Y -40.156,Z 176,A -15.1761,B 7.1287,C 0.2916,E1 7.2872,E2 467.1302} C_DIS
LIN {X 128.6173,Y -43.0944,Z 176,A -16.5058,B 7.1285,C 0.2957,E1 7.286,E2 468.4643} C_DIS
LIN {X 127.3833,Y -46.6195,Z 176,A -18.0311,B 7.1284,C 0.2991,E1 7.2846,E2 469.9847} C_DIS
LIN {X 126.2901,Y -49.5016,Z 176,A -19.3227,B 7.1282,C 0.3024,E1 7.2833,E2 471.2761} C_DIS
LIN {X 124.8862,Y -52.9472,Z 176,A -21.609,B 7.1275,C 0.3197,E1 7.2807,E2 473.653} C_DIS
LIN {X 122.5689,Y -58.1073,Z 176,A -23.0498,B 7.128,C 0.3087,E1 7.2791,E2 474.9779} C_DIS
LIN {X 121.4199,Y -60.4724,Z 176,A -24.2945,B 7.1277,C 0.314,E1 7.2776,E2 476.2405} C_DIS
LIN {X 119.5751,Y -64.0453,Z 176,A -26.0467,B 7.1275,C 0.3194,E1 7.2753,E2 478.0011} C_DIS
LIN {X 117.1611,Y -68.3623,Z 176,A -28.0365,B 7.1273,C 0.3229,E1 7.2726,E2 479.9804} C_DIS
LIN {X 114.844,Y -72.186,Z 176,A -29.7901,B 7.1273,C 0.3252,E1 7.27,E2 481.7189} C_DIS
LIN {X 113.4895,Y -74.2982,Z 176,A -31.0125,B 7.127,C 0.3307,E1 7.2681,E2 482.9627} C_DIS
LIN {X 110.2704,Y -78.9965,Z 176,A -33.1503,B 7.127,C 0.3317,E1 7.2648,E2 485.0692} C_DIS
LIN {X 108.3555,Y -81.6032,Z 176,A -34.7659,B 7.1266,C 0.3394,E1 7.262,E2 486.7175} C_DIS
LIN {X 106.22,Y -84.3641,Z 176,A -36.1783,B 7.1265,C 0.3417,E1 7.2596,E2 488.1235} C_DIS
LIN {X 103.3124,Y -87.9006,Z 176,A -38.0588,B 7.1263,C 0.3452,E1 7.2562,E2 489.9991} C_DIS
LIN {X 100.4546,Y -91.1529,Z 176,A -39.8583,B 7.1261,C 0.3487,E1 7.2529,E2 491.7967} C_DIS
LIN {X 97.3193,Y -94.4932,Z 176,A -41.7807,B 7.1259,C 0.3526,E1 7.2492,E2 493.7193} C_DIS
LIN {X 94.1923,Y -97.6107,Z 176,A -43.6128,B 7.1258,C 0.3559,E1 7.2455,E2 495.549} C_DIS
LIN {X 89.8839,Y -101.5916,Z 176,A -45.8368,B 7.1258,C 0.3564,E1 7.241,E2 497.7432} C_DIS
LIN {X 87.5213,Y -103.6349,Z 176,A -47.3964,B 7.1254,C 0.3632,E1 7.2376,E2 499.3344} C_DIS
LIN {X 82.8952,Y -107.3705,Z 176,A -49.8099,B 7.1252,C 0.3662,E1 7.2324,E2 501.7377} C_DIS
LIN {X 79.3196,Y -110.0386,Z 176,A -51.7409,B 7.125,C 0.3704,E1 7.228,E2 503.6763} C_DIS
LIN {X 75.8596,Y -112.4515,Z 176,A -53.4344,B 7.125,C 0.3719,E1 7.2241,E2 505.3602} C_DIS
LIN {X 72.3771,Y -114.7237,Z 176,A -55.2051,B 7.1248,C 0.375,E1 7.22,E2 507.1343} C_DIS
LIN {X 67.5936,Y -117.6064,Z 176,A -57.915,B 7.1243,C 0.3847,E1 7.2133,E2 509.8903} C_DIS
LIN {X 63.8638,Y -119.6726,Z 176,A -59.219,B 7.1246,C 0.3789,E1 7.2103,E2 511.1332} C_DIS
LIN {X 61.1607,Y -121.0742,Z 176,A -60.5166,B 7.1245,C 0.3809,E1 7.2071,E2 512.4332} C_DIS
LIN {X 57.7112,Y -122.7581,Z 176,A -62.129,B 7.1244,C 0.3829,E1 7.203,E2 514.0458} C_DIS
LIN {X 55.1574,Y -123.924,Z 176,A -63.2855,B 7.1244,C 0.3839,E1 7.2001,E2 515.1994} C_DIS
LIN {X 51.9782,Y -125.2909,Z 176,A -64.7491,B 7.1242,C 0.3857,E1 7.1963,E2 516.6644} C_DIS
LIN {X 48.222,Y -126.7855,Z 176,A -66.5309,B 7.124,C 0.389,E1 7.1916,E2 518.4569} C_DIS
LIN {X 44.6048,Y -128.1012,Z 176,A -68.0695,B 7.124,C 0.3892,E1 7.1876,E2 519.9856} C_DIS
LIN {X 41.1641,Y -129.2478,Z 176,A -69.539,B 7.124,C 0.3897,E1 7.1837,E2 521.4483} C_DIS
LIN {X 38.1145,Y -130.1797,Z 176,A -70.8674,B 7.124,C 0.3907,E1 7.1802,E2 522.7753} C_DIS
LIN {X 35.0924,Y -131.0268,Z 176,A -72.2101,B 7.1239,C 0.3921,E1 7.1765,E2 524.121} C_DIS
LIN {X 31.8801,Y -131.8452,Z 176,A -73.6025,B 7.1239,C 0.3931,E1 7.1728,E2 525.5133} C_DIS
LIN {X 28.3481,Y -132.6498,Z 176,A -75.1127,B 7.1238,C 0.3939,E1 7.1686,E2 527.022} C_DIS
LIN {X 25.0343,Y -133.3154,Z 176,A -76.5568,B 7.1238,C 0.3951,E1 7.1647,E2 528.4691} C_DIS
LIN {X 21.0808,Y -133.9972,Z 176,A -78.3183,B 7.1236,C 0.3972,E1 7.1598,E2 530.24} C_DIS
LIN {X 17.1735,Y -134.5542,Z 176,A -79.9648,B 7.1236,C 0.3977,E1 7.1552,E2 531.885} C_DIS
LIN {X 9.4752,Y -135.3143,Z 176,A -82.9718,B 7.1237,C 0.3948,E1 7.147,E2 534.8608} C_DIS
LIN {X 2.7599,Y -135.618,Z 176,A -86.0378,B 7.1235,C 0.3991,E1 7.1383,E2 537.9571} C_DIS
LIN {X 2.7599,Y -135.618,Z 176,A -86.0378,B 7.1235,C 0.3991,E1 7.1383,E2 537.9571} C_DIS
Enddeposition()
LIN {X 1.001,Y -136.5474,Z 176,A -86.4643,B 7.1002,C 0.3984,E1 7.1139,E2 538.3839} C_DIS
Startdeposition()
$VEL.CP = VEL_PRINT
LIN {X 8.1483,Y -136.3076,Z 176,A -83.0107,B 7.1006,C 0.3905,E1 7.1237,E2 534.8709} C_DIS
LIN {X 15.5761,Y -135.6607,Z 176,A -79.9505,B 7.1006,C 0.3905,E1 7.1322,E2 531.818} C_DIS
LIN {X 21.5097,Y -134.8472,Z 176,A -77.2898,B 7.1008,C 0.3867,E1 7.1396,E2 529.1367} C_DIS
LIN {X 25.376,Y -134.1722,Z 176,A -75.9077,B 7.1007,C 0.39,E1 7.1433,E2 527.7877} C_DIS
LIN {X 28.6202,Y -133.5176,Z 176,A -74.3973,B 7.1008,C 0.387,E1 7.1474,E2 526.2608} C_DIS
LIN {X 31.9988,Y -132.7483,Z 176,A -72.9742,B 7.1008,C 0.3864,E1 7.1513,E2 524.8407} C_DIS
LIN {X 35.2668,Y -131.9177,Z 176,A -71.5704,B 7.1009,C 0.3854,E1 7.1551,E2 523.4374} C_DIS
LIN {X 39.1087,Y -130.8324,Z 176,A -69.8054,B 7.1011,C 0.3823,E1 7.1599,E2 521.6597} C_DIS
LIN {X 42.6948,Y -129.7049,Z 176,A -68.2087,B 7.1011,C 0.3804,E1 7.1641,E2 520.0593} C_DIS
LIN {X 46.6663,Y -128.3292,Z 176,A -66.5049,B 7.1012,C 0.3796,E1 7.1686,E2 518.3619} C_DIS
LIN {X 50.6456,Y -126.8116,Z 176,A -64.7922,B 7.1012,C 0.3788,E1 7.173,E2 516.6575} C_DIS
LIN {X 53.9458,Y -125.4428,Z 176,A -63.2618,B 7.1014,C 0.3764,E1 7.177,E2 515.1219} C_DIS
LIN {X 56.7836,Y -124.185,Z 176,A -62.0411,B 7.1014,C 0.3761,E1 7.18,E2 513.9108} C_DIS
LIN {X 59.5407,Y -122.8879,Z 176,A -60.5951,B 7.1017,C 0.3715,E1 7.1837,E2 512.4422} C_DIS
LIN {X 63.3012,Y -120.9915,Z 176,A -59.1325,B 7.1015,C 0.3743,E1 7.1873,E2 511.0173} C_DIS
LIN {X 69.7136,Y -117.4163,Z 176,A -55.7009,B 7.1021,C 0.3635,E1 7.1957,E2 507.5381} C_DIS
LIN {X 74.2075,Y -114.6289,Z 176,A -53.6696,B 7.1021,C 0.3632,E1 7.2005,E2 505.5293} C_DIS
LIN {X 77.4799,Y -112.443,Z 176,A -52.08,B 7.1021,C 0.3615,E1 7.2041,E2 503.9461} C_DIS
LIN {X 81.0557,Y -109.8934,Z 176,A -50.2532,B 7.1023,C 0.3585,E1 7.2082,E2 502.1198} C_DIS
LIN {X 84.4616,Y -107.2976,Z 176,A -48.3863,B 7.1025,C 0.3539,E1 7.2124,E2 500.2422} C_DIS
LIN {X 88.1392,Y -104.2983,Z 176,A -46.3929,B 7.1027,C 0.3501,E1 7.2167,E2 498.2467} C_DIS
LIN {X 92.2482,Y -100.6818,Z 176,A -44.2041,B 7.1029,C 0.3474,E1 7.2212,E2 496.0698} C_DIS
LIN {X 95.7034,Y -97.4032,Z 176,A -42.2643,B 7.103,C 0.3444,E1 7.2251,E2 494.1357} C_DIS
LIN {X 98.6948,Y -94.3707,Z 176,A -40.5192,B 7.1032,C 0.3413,E1 7.2285,E2 492.3943} C_DIS
LIN {X 101.5109,Y -91.3353,Z 176,A -38.7691,B 7.1034,C 0.3373,E1 7.2318,E2 490.641} C_DIS
LIN {X 104.4746,Y -87.9296,Z 176,A -36.9055,B 7.1035,C 0.3336,E1 7.2351,E2 488.7795} C_DIS
LIN {X 107.0631,Y -84.7593,Z 176,A -35.216,B 7.1037,C 0.3301,E1 7.2381,E2 487.092} C_DIS
LIN {X 109.5835,Y -81.4738,Z 176,A -33.5901,B 7.1037,C 0.3281,E1 7.2408,E2 485.4788} C_DIS
LIN {X 111.6306,Y -78.6456,Z 176,A -32.039,B 7.104,C 0.323,E1 7.2433,E2 483.9151} C_DIS
LIN {X 114.2865,Y -74.7347,Z 176,A -30.3567,B 7.104,C 0.3237,E1 7.2459,E2 482.2696} C_DIS
LIN {X 116.7279,Y -70.86,Z 176,A -28.3199,B 7.1043,C 0.3168,E1 7.2489,E2 480.2162} C_DIS
LIN {X 118.8041,Y -67.3219,Z 176,A -26.5242,B 7.1045,C 0.3111,E1 7.2514,E2 478.4093} C_DIS
LIN {X 120.8033,Y -63.6596,Z 176,A -25.1361,B 7.1045,C 0.3133,E1 7.2532,E2 477.0658} C_DIS
LIN {X 122.3533,Y -60.6275,Z 176,A -23.6559,B 7.1046,C 0.3086,E1 7.2551,E2 475.5778} C_DIS
LIN {X 123.6122,Y -58.0224,Z 176,A -22.2194,B 7.105,C 0.3013,E1 7.2569,E2 474.1117} C_DIS
LIN {X 125.6975,Y -53.3548,Z 176,A -20.1165,B 7.1052,C 0.2964,E1 7.2592,E2 472.0121} C_DIS
LIN {X 127.1499,Y -49.7896,Z 176,A -18.7289,B 7.1052,C 0.2962,E1 7.2606,E2 470.652} C_DIS
LIN {X 128.3049,Y -46.7337,Z 176,A -17.4489,B 7.1052,C 0.2942,E1 7.2619,E2 469.3823} C_DIS
LIN {X 129.4433,Y -43.4806,Z 176,A -15.7919,B 7.1056,C 0.2863,E1 7.2634,E2 467.697} C_DIS
LIN {X 130.4605,Y -40.3263,Z 176,A -14.4256,B 7.1057,C 0.2829,E1 7.2645,E2 466.3326} C_DIS
LIN {X 131.7177,Y -36.015,Z 176,A -12.6788,B 7.1058,C 0.2802,E1 7.2658,E2 464.6016} C_DIS
LIN {X 132.7985,Y -31.7903,Z 176,A -10.8421,B 7.106,C 0.275,E1 7.2671,E2 462.7623} C_DIS
LIN {X 133.7371,Y -27.5782,Z 176,A -9.0815,B 7.1062,C 0.2708,E1 7.2681,E2 461.0064} C_DIS
LIN {X 134.3739,Y -24.2851,Z 176,A -7.8327,B 7.1062,C 0.2698,E1 7.2687,E2 459.7764} C_DIS
LIN {X 134.8117,Y -21.7354,Z 176,A -6.5084,B 7.1065,C 0.2622,E1 7.2694,E2 458.4208} C_DIS
LIN {X 135.4016,Y -17.677,Z 176,A -4.9439,B 7.1065,C 0.2602,E1 7.2699,E2 456.8746} C_DIS
LIN {X 135.8424,Y -13.9075,Z 176,A -2.9222,B 7.107,C 0.2476,E1 7.2706,E2 454.7968} C_DIS
LIN {X 136.2126,Y -9.6096,Z 176,A -1.1088,B 7.1072,C 0.2423,E1 7.2709,E2 452.9814} C_DIS
LIN {X 136.4598,Y -4.9945,Z 176,A 0.3893,B 7.1072,C 0.2451,E1 7.2711,E2 451.5379} C_DIS
LIN {X 136.5504,Y -0.6257,Z 176,A 2.0921,B 7.1072,C 0.2422,E1 7.2711,E2 449.8501} C_DIS
LIN {X 136.4977,Y 3.8083,Z 176,A 3.9257,B 7.1074,C 0.2374,E1 7.2711,E2 448.0184} C_DIS
LIN {X 136.1654,Y 10.2557,Z 176,A 6.6302,B 7.1076,C 0.2297,E1 7.2706,E2 445.3123} C_DIS
LIN {X 135.8327,Y 13.9979,Z 176,A 8.176,B 7.1077,C 0.2258,E1 7.2702,E2 443.7691} C_DIS
LIN {X 135.3824,Y 17.8234,Z 176,A 9.581,B 7.1077,C 0.2251,E1 7.2697,E2 442.3895} C_DIS
LIN {X 134.9504,Y 20.8433,Z 176,A 11.0031,B 7.108,C 0.2189,E1 7.2691,E2 440.9485} C_DIS
LIN {X 134.1813,Y 25.3285,Z 176,A 12.8039,B 7.108,C 0.2155,E1 7.2682,E2 439.16} C_DIS
LIN {X 133.4117,Y 29.1108,Z 176,A 14.4755,B 7.1082,C 0.21,E1 7.2672,E2 437.4807} C_DIS
LIN {X 132.5816,Y 32.6903,Z 176,A 16.0076,B 7.1083,C 0.2059,E1 7.2662,E2 435.9488} C_DIS
LIN {X 131.5669,Y 36.5544,Z 176,A 17.5168,B 7.1083,C 0.2043,E1 7.2651,E2 434.4594} C_DIS
LIN {X 130.6289,Y 39.776,Z 176,A 18.9613,B 7.1085,C 0.1998,E1 7.264,E2 433.0094} C_DIS
LIN {X 129.5357,Y 43.2031,Z 176,A 20.389,B 7.1085,C 0.1972,E1 7.2628,E2 431.5909} C_DIS
LIN {X 128.4404,Y 46.3579,Z 176,A 22.1642,B 7.1089,C 0.1865,E1 7.261,E2 429.7677} C_DIS
LIN {X 127.0405,Y 50.0708,Z 176,A 23.5958,B 7.1089,C 0.1865,E1 7.2596,E2 428.3646} C_DIS
LIN {X 125.5267,Y 53.7516,Z 176,A 25.0985,B 7.1089,C 0.1851,E1 7.258,E2 426.8818} C_DIS
LIN {X 124.0114,Y 57.1591,Z 176,A 26.5414,B 7.1089,C 0.1832,E1 7.2563,E2 425.4533} C_DIS
LIN {X 122.7666,Y 59.7896,Z 176,A 27.8845,B 7.1091,C 0.1779,E1 7.2547,E2 424.0943} C_DIS
LIN {X 121.113,Y 63.0699,Z 176,A 29.3166,B 7.1091,C 0.1759,E1 7.2529,E2 422.675} C_DIS
LIN {X 119.1404,Y 66.7242,Z 176,A 31.08,B 7.1093,C 0.1712,E1 7.2505,E2 420.9082} C_DIS
LIN {X 116.9138,Y 70.5528,Z 176,A 32.931,B 7.1093,C 0.1668,E1 7.2479,E2 419.0572} C_DIS
LIN {X 114.4105,Y 74.5439,Z 176,A 34.8457,B 7.1095,C 0.1631,E1 7.245,E2 417.1494} C_DIS
LIN {X 112.0169,Y 78.0944,Z 176,A 36.5691,B 7.1095,C 0.1602,E1 7.2423,E2 415.4344} C_DIS
LIN {X 109.7258,Y 81.2827,Z 176,A 38.2284,B 7.1096,C 0.1562,E1 7.2396,E2 413.7729} C_DIS
LIN {X 107.254,Y 84.5171,Z 176,A 40.0311,B 7.1097,C 0.1506,E1 7.2364,E2 411.9577} C_DIS
LIN {X 104.1464,Y 88.3179,Z 176,A 41.9767,B 7.1097,C 0.1481,E1 7.233,E2 410.0256} C_DIS
LIN {X 101.0833,Y 91.8078,Z 176,A 43.617,B 7.1097,C 0.1494,E1 7.23,E2 408.423} C_DIS
LIN {X 98.1991,Y 94.8865,Z 176,A 45.6383,B 7.1099,C 0.1413,E1 7.2261,E2 406.3701} C_DIS
LIN {X 95.3347,Y 97.7648,Z 176,A 47.5063,B 7.11,C 0.135,E1 7.2223,E2 404.4811} C_DIS
LIN {X 92.9672,Y 100.0182,Z 176,A 48.6384,B 7.11,C 0.1366,E1 7.2201,E2 403.3786} C_DIS
LIN {X 89.5641,Y 103.0769,Z 176,A 50.5584,B 7.11,C 0.1329,E1 7.216,E2 401.4581} C_DIS
LIN {X 86.0649,Y 106.0167,Z 176,A 52.4859,B 7.1101,C 0.1292,E1 7.2119,E2 399.529} C_DIS
LIN {X 82.4441,Y 108.8555,Z 176,A 54.3743,B 7.1101,C 0.1266,E1 7.2077,E2 397.6456} C_DIS
LIN {X 78.8771,Y 111.4673,Z 176,A 56.1812,B 7.1102,C 0.1243,E1 7.2036,E2 395.8444} C_DIS
LIN {X 75.5791,Y 113.7294,Z 176,A 57.8724,B 7.1102,C 0.1214,E1 7.1997,E2 394.1514} C_DIS
LIN {X 71.715,Y 116.205,Z 176,A 59.7839,B 7.1103,C 0.1187,E1 7.1952,E2 392.2415} C_DIS
LIN {X 67.805,Y 118.5286,Z 176,A 61.6372,B 7.1103,C 0.1169,E1 7.1907,E2 390.395} C_DIS
LIN {X 63.9104,Y 120.6717,Z 176,A 63.3989,B 7.1103,C 0.1161,E1 7.1864,E2 388.6461} C_DIS
LIN {X 60.6515,Y 122.3414,Z 176,A 64.9893,B 7.1104,C 0.1132,E1 7.1825,E2 387.049} C_DIS
LIN {X 57.3739,Y 123.9121,Z 176,A 66.4251,B 7.1104,C 0.1128,E1 7.1789,E2 385.6243} C_DIS
LIN {X 54.2997,Y 125.2898,Z 176,A 67.7414,B 7.1104,C 0.1128,E1 7.1755,E2 384.32} C_DIS
LIN {X 49.2678,Y 127.3527,Z 176,A 70.1711,B 7.1104,C 0.1079,E1 7.1692,E2 381.8725} C_DIS
LIN {X 44.8627,Y 128.9703,Z 176,A 72.0296,B 7.1105,C 0.1078,E1 7.1643,E2 380.0278} C_DIS
LIN {X 41.6967,Y 130.0285,Z 176,A 73.4439,B 7.1105,C 0.1063,E1 7.1606,E2 378.6121} C_DIS
LIN {X 37.7506,Y 131.23,Z 176,A 75.2589,B 7.1105,C 0.1035,E1 7.1557,E2 376.7872} C_DIS
LIN {X 33.8389,Y 132.2914,Z 176,A 76.8399,B 7.1105,C 0.1042,E1 7.1515,E2 375.2212} C_DIS
LIN {X 30.6816,Y 133.0592,Z 176,A 78.183,B 7.1105,C 0.1036,E1 7.1478,E2 373.8809} C_DIS
LIN {X 27.8013,Y 133.6917,Z 176,A 79.5814,B 7.1106,C 0.1003,E1 7.1439,E2 372.4631} C_DIS
LIN {X 23.4182,Y 134.529,Z 176,A 81.4322,B 7.1106,C 0.0997,E1 7.1389,E2 370.6156} C_DIS
LIN {X 18.712,Y 135.2638,Z 176,A 83.5439,B 7.1106,C 0.0971,E1 7.133,E2 368.4905} C_DIS
LIN {X 14.009,Y 135.8315,Z 176,A 85.5509,B 7.1106,C 0.0961,E1 7.1274,E2 366.4819} C_DIS
LIN {X 8.7448,Y 136.2709,Z 176,A 87.4069,B 7.1106,C 0.1012,E1 7.1224,E2 364.671} C_DIS
LIN {X 3.0979,Y 136.5174,Z 176,A 90.0066,B 7.1106,C 0.0975,E1 7.115,E2 362.0444} C_DIS
LIN {X -3.8007,Y 136.4979,Z 176,A 92.7926,B 7.1106,C 0.0992,E1 7.1073,E2 359.273} C_DIS
LIN {X -8.0828,Y 136.3117,Z 176,A 94.6263,B 7.1106,C 0.0989,E1 7.1022,E2 357.4359} C_DIS
LIN {X -12.1815,Y 136.008,Z 176,A 96.4439,B 7.1106,C 0.0979,E1 7.0971,E2 355.6078} C_DIS
LIN {X -15.7763,Y 135.6368,Z 176,A 97.7359,B 7.1106,C 0.1017,E1 7.0936,E2 354.3441} C_DIS
LIN {X -19.1766,Y 135.1974,Z 176,A 99.2559,B 7.1106,C 0.1011,E1 7.0893,E2 352.815} C_DIS
LIN {X -22.7013,Y 134.6505,Z 176,A 100.7603,B 7.1106,C 0.1016,E1 7.0852,E2 351.3105} C_DIS
LIN {X -26.8577,Y 133.8837,Z 176,A 102.5686,B 7.1106,C 0.1021,E1 7.0802,E2 349.4989} C_DIS
LIN {X -29.9079,Y 133.2359,Z 176,A 103.888,B 7.1106,C 0.1027,E1 7.0766,E2 348.1791} C_DIS
LIN {X -33.4468,Y 132.3909,Z 176,A 105.3797,B 7.1106,C 0.1043,E1 7.0726,E2 346.6926} C_DIS
LIN {X -37.0732,Y 131.4218,Z 176,A 107.0787,B 7.1106,C 0.1037,E1 7.068,E2 344.9794} C_DIS
LIN {X -41.4161,Y 130.1181,Z 176,A 108.8815,B 7.1106,C 0.1067,E1 7.0632,E2 343.1901} C_DIS
LIN {X -45.8706,Y 128.6161,Z 176,A 110.9134,B 7.1106,C 0.1077,E1 7.0578,E2 341.1524} C_DIS
LIN {X -51.1149,Y 126.6224,Z 176,A 113.2279,B 7.1105,C 0.1107,E1 7.0518,E2 338.8444} C_DIS
LIN {X -54.0669,Y 125.3904,Z 176,A 114.565,B 7.1105,C 0.1123,E1 7.0484,E2 337.5089} C_DIS
LIN {X -57.7367,Y 123.7443,Z 176,A 116.6443,B 7.1105,C 0.1088,E1 7.043,E2 335.3828} C_DIS
LIN {X -61.0259,Y 122.1567,Z 176,A 117.9857,B 7.1105,C 0.1135,E1 7.0397,E2 334.0662} C_DIS
LIN {X -64.973,Y 120.1048,Z 176,A 119.8529,B 7.1104,C 0.116,E1 7.0351,E2 332.2004} C_DIS
LIN {X -70.7431,Y 116.7987,Z 176,A 122.64,B 7.1104,C 0.1201,E1 7.0284,E2 329.416} C_DIS
LIN {X -74.6326,Y 114.3529,Z 176,A 124.5407,B 7.1102,C 0.1234,E1 7.0239,E2 327.5201} C_DIS
LIN {X -77.0568,Y 112.7334,Z 176,A 126.6117,B 7.1104,C 0.1139,E1 7.019,E2 325.3455} C_DIS
LIN {X -82.2254,Y 109.0206,Z 176,A 128.2,B 7.1101,C 0.1331,E1 7.0157,E2 323.8931} C_DIS
LIN {X -84.8084,Y 107.0239,Z 176,A 129.9501,B 7.1101,C 0.1305,E1 7.0117,E2 322.0976} C_DIS
LIN {X -88.3917,Y 104.0837,Z 176,A 131.6083,B 7.11,C 0.1378,E1 7.0082,E2 320.4762} C_DIS
LIN {X -91.0721,Y 101.7466,Z 176,A 133.3972,B 7.11,C 0.1368,E1 7.0044,E2 318.6523} C_DIS
LIN {X -94.121,Y 98.9335,Z 176,A 135.2447,B 7.11,C 0.1388,E1 7.0006,E2 316.7933} C_DIS
LIN {X -97.7101,Y 95.3905,Z 176,A 137.1956,B 7.1098,C 0.1453,E1 6.9968,E2 314.8646} C_DIS
LIN {X -100.8133,Y 92.1052,Z 176,A 139.2684,B 7.1098,C 0.147,E1 6.9928,E2 312.7718} C_DIS
LIN {X -102.9339,Y 89.728,Z 176,A 140.5996,B 7.1098,C 0.15,E1 6.9904,E2 311.4425} C_DIS
LIN {X -105.7762,Y 86.3592,Z 176,A 142.4748,B 7.1097,C 0.1537,E1 6.987,E2 309.5659} C_DIS
LIN {X -109.4809,Y 81.6115,Z 176,A 145.0502,B 7.1095,C 0.1589,E1 6.9827,E2 306.9869} C_DIS
LIN {X -112.1226,Y 77.9425,Z 176,A 146.9565,B 7.1095,C 0.1632,E1 6.9796,E2 305.0813} C_DIS
LIN {X -114.6711,Y 74.1425,Z 176,A 148.9485,B 7.1094,C 0.167,E1 6.9765,E2 303.0821} C_DIS
LIN {X -117.2322,Y 70.0223,Z 176,A 151.7318,B 7.1094,C 0.1625,E1 6.9724,E2 300.2078} C_DIS
LIN {X -120.2186,Y 64.7612,Z 176,A 153.6876,B 7.1091,C 0.1763,E1 6.9699,E2 298.3271} C_DIS
LIN {X -121.9918,Y 61.3548,Z 176,A 155.1412,B 7.109,C 0.1824,E1 6.9681,E2 296.8945} C_DIS
LIN {X -123.7782,Y 57.6635,Z 176,A 156.9474,B 7.1089,C 0.1858,E1 6.9659,E2 295.0793} C_DIS
LIN {X -125.1528,Y 54.6166,Z 176,A 158.2714,B 7.1088,C 0.1905,E1 6.9644,E2 293.7664} C_DIS
LIN {X -126.4684,Y 51.4972,Z 176,A 159.7861,B 7.1088,C 0.1931,E1 6.9628,E2 292.2414} C_DIS
LIN {X -130.2094,Y 41.1303,Z 176,A 164.3007,B 7.1083,C 0.2071,E1 6.9586,E2 287.7452} C_DIS
LIN {X -131.3793,Y 37.2249,Z 176,A 166.1271,B 7.1083,C 0.2104,E1 6.9571,E2 285.906} C_DIS
LIN {X -132.3111,Y 33.7615,Z 176,A 167.8007,B 7.1082,C 0.2125,E1 6.9559,E2 284.2129} C_DIS
LIN {X -133.2952,Y 29.6483,Z 176,A 169.7102,B 7.1081,C 0.2158,E1 6.9547,E2 282.2884} C_DIS
LIN {X -134.1039,Y 25.7335,Z 176,A 171.2812,B 7.1079,C 0.2219,E1 6.9539,E2 280.7321} C_DIS
LIN {X -134.7965,Y 21.8264,Z 176,A 173.0991,B 7.1078,C 0.2247,E1 6.953,E2 278.8967} C_DIS
LIN {X -135.3762,Y 17.8707,Z 176,A 174.7063,B 7.1076,C 0.2304,E1 6.9524,E2 277.2997} C_DIS
LIN {X -135.7915,Y 14.3811,Z 176,A 176.2485,B 7.1075,C 0.2338,E1 6.9519,E2 275.7504} C_DIS
LIN {X -136.1715,Y 10.1716,Z 176,A 178.0765,B 7.1073,C 0.2382,E1 6.9515,E2 273.9172} C_DIS
LIN {X -136.4276,Y 5.8195,Z 176,A 179.9229,B 7.1072,C 0.2432,E1 6.9512,E2 272.0702} C_DIS
LIN {X -136.5346,Y 2.1067,Z 176,A -178.4971,B 7.107,C 0.2474,E1 6.9512,E2 270.4889} C_DIS
LIN {X -136.5343,Y -2.1288,Z 176,A -176.7095,B 7.1069,C 0.2524,E1 6.9512,E2 268.7014} C_DIS
LIN {X -136.4378,Y -5.5572,Z 176,A -175.1475,B 7.1068,C 0.255,E1 6.9513,E2 267.1252} C_DIS
LIN {X -136.1932,Y -9.8749,Z 176,A -173.3795,B 7.1066,C 0.2608,E1 6.9516,E2 265.3645} C_DIS
LIN {X -135.8838,Y -13.486,Z 176,A -171.699,B 7.1065,C 0.2631,E1 6.9521,E2 263.6652} C_DIS
LIN {X -135.4668,Y -17.1796,Z 176,A -170.1489,B 7.1063,C 0.2677,E1 6.9526,E2 262.1176} C_DIS
LIN {X -134.9395,Y -20.9137,Z 176,A -168.6248,B 7.1061,C 0.2729,E1 6.9532,E2 260.602} C_DIS
LIN {X -134.3677,Y -24.3196,Z 176,A -167.1103,B 7.106,C 0.2762,E1 6.954,E2 259.0804} C_DIS
LIN {X -133.5214,Y -28.6028,Z 176,A -165.2707,B 7.1058,C 0.2812,E1 6.955,E2 257.2411} C_DIS
LIN {X -132.7904,Y -31.8242,Z 176,A -163.8284,B 7.1057,C 0.2843,E1 6.9559,E2 255.7928} C_DIS
LIN {X -129.8874,Y -42.1383,Z 176,A -159.6454,B 7.105,C 0.3007,E1 6.9591,E2 251.6526} C_DIS
LIN {X -128.3912,Y -46.4944,Z 176,A -157.2835,B 7.105,C 0.3005,E1 6.9613,E2 249.2382} C_DIS
LIN {X -126.9309,Y -50.3498,Z 176,A -155.4253,B 7.1049,C 0.3034,E1 6.9632,E2 247.3649} C_DIS
LIN {X -125.4544,Y -53.9188,Z 176,A -153.8623,B 7.1047,C 0.3084,E1 6.9649,E2 245.81} C_DIS
LIN {X -124.1342,Y -56.8935,Z 176,A -152.5999,B 7.1044,C 0.3132,E1 6.9663,E2 244.5615} C_DIS
LIN {X -122.5884,Y -60.1508,Z 176,A -150.9485,B 7.1044,C 0.3153,E1 6.9683,E2 242.8935} C_DIS
LIN {X -120.9019,Y -63.4719,Z 176,A -149.3959,B 7.1042,C 0.3194,E1 6.9703,E2 241.343} C_DIS
LIN {X -118.2955,Y -68.2111,Z 176,A -146.9348,B 7.104,C 0.3225,E1 6.9737,E2 238.8589} C_DIS
LIN {X -115.9138,Y -72.1838,Z 176,A -144.9855,B 7.1038,C 0.3271,E1 6.9765,E2 236.9098} C_DIS
LIN {X -113.1285,Y -76.4752,Z 176,A -142.837,B 7.1036,C 0.3321,E1 6.9798,E2 234.7621} C_DIS
LIN {X -110.711,Y -79.9353,Z 176,A -141.2109,B 7.1033,C 0.338,E1 6.9824,E2 233.1551} C_DIS
LIN {X -108.1811,Y -83.3277,Z 176,A -139.1664,B 7.1033,C 0.3385,E1 6.9859,E2 231.0772} C_DIS
LIN {X -105.4303,Y -86.782,Z 176,A -137.2715,B 7.1031,C 0.3419,E1 6.9893,E2 229.1776} C_DIS
LIN {X -102.4783,Y -90.2484,Z 176,A -135.0029,B 7.1031,C 0.3411,E1 6.9935,E2 226.8639} C_DIS
LIN {X -99.7056,Y -93.3019,Z 176,A -133.6111,B 7.1028,C 0.3492,E1 6.9961,E2 225.516} C_DIS
LIN {X -96.5959,Y -96.5188,Z 176,A -131.672,B 7.1026,C 0.3521,E1 6.9999,E2 223.5695} C_DIS
LIN {X -93.3548,Y -99.6572,Z 176,A -129.7891,B 7.1025,C 0.3558,E1 7.0037,E2 221.6884} C_DIS
LIN {X -90.1175,Y -102.594,Z 176,A -127.8978,B 7.1023,C 0.3584,E1 7.0077,E2 219.7901} C_DIS
LIN {X -86.6617,Y -105.5289,Z 176,A -125.9873,B 7.1022,C 0.3616,E1 7.0118,E2 217.879} C_DIS
LIN {X -83.1804,Y -108.2941,Z 176,A -124.0902,B 7.102,C 0.3643,E1 7.016,E2 215.9781} C_DIS
LIN {X -79.6758,Y -110.898,Z 176,A -122.1333,B 7.102,C 0.3655,E1 7.0204,E2 214.0054} C_DIS
LIN {X -75.4162,Y -113.8379,Z 176,A -120.027,B 7.1017,C 0.3697,E1 7.0253,E2 211.9077} C_DIS
LIN {X -71.8916,Y -116.0956,Z 176,A -118.2995,B 7.1016,C 0.3726,E1 7.0293,E2 210.1839} C_DIS
LIN {X -68.0337,Y -118.3981,Z 176,A -116.3591,B 7.1016,C 0.3744,E1 7.034,E2 208.2366} C_DIS
LIN {X -64.1733,Y -120.5336,Z 176,A -114.4743,B 7.1014,C 0.3763,E1 7.0387,E2 206.3474} C_DIS
LIN {X -60.6934,Y -122.3208,Z 176,A -112.9486,B 7.1012,C 0.3799,E1 7.0424,E2 204.8364} C_DIS
LIN {X -57.5604,Y -123.8258,Z 176,A -111.4899,B 7.1012,C 0.3815,E1 7.0461,E2 203.3775} C_DIS
LIN {X -52.0211,Y -126.2545,Z 176,A -108.9337,B 7.101,C 0.3839,E1 7.0527,E2 200.8189} C_DIS
LIN {X -48.9483,Y -127.4769,Z 176,A -107.4216,B 7.101,C 0.3833,E1 7.0567,E2 199.2906} C_DIS
LIN {X -45.3127,Y -128.8143,Z 176,A -105.8921,B 7.1009,C 0.3862,E1 7.0607,E2 197.7732} C_DIS
LIN {X -40.6694,Y -130.3555,Z 176,A -103.7049,B 7.1009,C 0.3857,E1 7.0665,E2 195.5684} C_DIS
LIN {X -37.0372,Y -131.4318,Z 176,A -102.2478,B 7.1007,C 0.3888,E1 7.0704,E2 194.1279} C_DIS
LIN {X -33.881,Y -132.2807,Z 176,A -100.8717,B 7.1007,C 0.3896,E1 7.0741,E2 192.7509} C_DIS
LIN {X -30.819,Y -133.0278,Z 176,A -99.4497,B 7.1007,C 0.3888,E1 7.078,E2 191.3157} C_DIS
LIN {X -26.7895,Y -133.8976,Z 176,A -97.6607,B 7.1007,C 0.3887,E1 7.0829,E2 189.5186} C_DIS
LIN {X -21.7406,Y -134.8108,Z 176,A -94.3876,B 7.1016,C 0.3719,E1 7.0924,E2 186.0991} C_DIS
LIN {X -13.4274,Y -135.8894,Z 176,A -92.2552,B 7.1004,C 0.3945,E1 7.0978,E2 184.1455} C_DIS
LIN {X -9.6762,Y -136.2077,Z 176,A -90.3193,B 7.1007,C 0.389,E1 7.1033,E2 182.1631} C_DIS
LIN {X -5.7127,Y -136.4318,Z 176,A -88.5017,B 7.1009,C 0.3866,E1 7.1084,E2 180.3251} C_DIS
LIN {X -2.0635,Y -136.5354,Z 176,A -87.319,B 7.1006,C 0.3921,E1 7.1116,E2 179.1869} C_DIS
LIN {X 1.001,Y -136.5474,Z 176,A -86.4616,B 7.1002,C 0.3988,E1 7.1139,E2 178.3839} C_DIS
Enddeposition()
LIN {X 1.001,Y -136.5474,Z 176,A -86.4616,B 7.1002,C 0.3988,E1 7.1139,E2 178.3839} C_DIS
Startdeposition()
$VEL.CP = VEL_PRINT
LIN {X -1.1461,Y -137.4523,Z 176,A -87.5371,B 7.0779,C 0.4059,E1 7.0889,E2 179.5227} C_DIS
LIN {X -4.261,Y -137.3911,Z 176,A -88.8313,B 7.0779,C 0.4059,E1 7.0852,E2 180.8168} C_DIS
LIN {X -7.3475,Y -137.2607,Z 176,A -90.1221,B 7.0779,C 0.4059,E1 7.0816,E2 182.1085} C_DIS
LIN {X -10.7874,Y -137.0347,Z 176,A -91.5412,B 7.0779,C 0.4055,E1 7.0777,E2 183.526} C_DIS
LIN {X -13.3679,Y -136.805,Z 176,A -92.678,B 7.0779,C 0.4062,E1 7.0745,E2 184.6705} C_DIS
LIN {X -17.0709,Y -136.3945,Z 176,A -94.1825,B 7.0779,C 0.4051,E1 7.0703,E2 186.1694} C_DIS
LIN {X -19.7037,Y -136.037,Z 176,A -95.3166,B 7.0779,C 0.4052,E1 7.0672,E2 187.3072} C_DIS
LIN {X -23.0807,Y -135.5054,Z 176,A -96.712,B 7.078,C 0.4043,E1 7.0634,E2 188.6994} C_DIS
LIN {X -26.0369,Y -134.968,Z 176,A -98.0112,B 7.078,C 0.4045,E1 7.0598,E2 190.005} C_DIS
LIN {X -29.8083,Y -134.1877,Z 176,A -99.5961,B 7.078,C 0.4034,E1 7.0555,E2 191.5877} C_DIS
LIN {X -32.673,Y -133.5174,Z 176,A -100.8296,B 7.0781,C 0.4028,E1 7.0521,E2 192.8224} C_DIS
LIN {X -36.2195,Y -132.601,Z 176,A -102.3653,B 7.0781,C 0.402,E1 7.048,E2 194.3596} C_DIS
LIN {X -39.4257,Y -131.6833,Z 176,A -103.7646,B 7.0782,C 0.4012,E1 7.0442,E2 195.7604} C_DIS
LIN {X -42.289,Y -130.7901,Z 176,A -105.0236,B 7.0782,C 0.4004,E1 7.0408,E2 197.0207} C_DIS
LIN {X -45.4374,Y -129.7297,Z 176,A -106.4479,B 7.0782,C 0.3998,E1 7.0371,E2 198.4503} C_DIS
LIN {X -48.4751,Y -128.625,Z 176,A -107.7997,B 7.0783,C 0.3987,E1 7.0335,E2 199.8028} C_DIS
LIN {X -52.1822,Y -127.1688,Z 176,A -109.4492,B 7.0784,C 0.3969,E1 7.0292,E2 201.4513} C_DIS
LIN {X -55.3382,Y -125.8275,Z 176,A -110.8909,B 7.0785,C 0.3956,E1 7.0255,E2 202.8947} C_DIS
LIN {X -58.1114,Y -124.5689,Z 176,A -112.1711,B 7.0785,C 0.3944,E1 7.0223,E2 204.1763} C_DIS
LIN {X -61.5873,Y -122.8897,Z 176,A -113.7958,B 7.0787,C 0.3928,E1 7.0182,E2 205.8032} C_DIS
LIN {X -64.3474,Y -121.4652,Z 176,A -115.1012,B 7.0787,C 0.3913,E1 7.015,E2 207.1098} C_DIS
LIN {X -67.7302,Y -119.6139,Z 176,A -116.8396,B 7.0787,C 0.3911,E1 7.0107,E2 208.865} C_DIS
LIN {X -71.5037,Y -117.3972,Z 176,A -118.571,B 7.079,C 0.3873,E1 7.0066,E2 210.5845} C_DIS
LIN {X -74.5755,Y -115.4698,Z 176,A -120.2115,B 7.079,C 0.3869,E1 7.0027,E2 212.2414} C_DIS
LIN {X -78.2979,Y -112.9787,Z 176,A -122.0834,B 7.0791,C 0.3841,E1 6.9984,E2 214.1138} C_DIS
LIN {X -81.5869,Y -110.6269,Z 176,A -123.6858,B 7.0794,C 0.3803,E1 6.9948,E2 215.7054} C_DIS
LIN {X -84.7062,Y -108.2571,Z 176,A -125.4431,B 7.0794,C 0.3793,E1 6.9908,E2 217.4783} C_DIS
LIN {X -88.1549,Y -105.4678,Z 176,A -127.3024,B 7.0796,C 0.3762,E1 6.9868,E2 219.3386} C_DIS
LIN {X -91.4685,Y -102.6075,Z 176,A -129.1807,B 7.0797,C 0.3736,E1 6.9829,E2 221.2233} C_DIS
LIN {X -94.5124,Y -99.8106,Z 176,A -130.8164,B 7.0799,C 0.3692,E1 6.9795,E2 222.8475} C_DIS
LIN {X -97.0642,Y -97.3308,Z 176,A -132.3433,B 7.0801,C 0.3669,E1 6.9765,E2 224.3796} C_DIS
LIN {X -99.6812,Y -94.6495,Z 176,A -133.9533,B 7.0801,C 0.3644,E1 6.9734,E2 225.9952} C_DIS
LIN {X -102.5643,Y -91.5167,Z 176,A -135.6999,B 7.0804,C 0.3604,E1 6.9701,E2 227.7377} C_DIS
LIN {X -104.8909,Y -88.8405,Z 176,A -137.2789,B 7.0804,C 0.3586,E1 6.9672,E2 229.329} C_DIS
LIN {X -107.7086,Y -85.4026,Z 176,A -139.1115,B 7.0807,C 0.3543,E1 6.964,E2 231.1584} C_DIS
LIN {X -109.9874,Y -82.4478,Z 176,A -140.7847,B 7.0807,C 0.3524,E1 6.9611,E2 232.8459} C_DIS
LIN {X -112.6124,Y -78.8243,Z 176,A -142.6883,B 7.081,C 0.3486,E1 6.9581,E2 234.7535} C_DIS
LIN {X -115.0523,Y -75.2187,Z 176,A -144.409,B 7.0812,C 0.3432,E1 6.9554,E2 236.4615} C_DIS
LIN {X -117.2155,Y -71.7999,Z 176,A -146.1729,B 7.0814,C 0.3402,E1 6.9528,E2 238.2345} C_DIS
LIN {X -119.1809,Y -68.4893,Z 176,A -147.7564,B 7.0816,C 0.336,E1 6.9506,E2 239.8144} C_DIS
LIN {X -120.969,Y -65.2782,Z 176,A -149.4344,B 7.0816,C 0.3341,E1 6.9483,E2 241.5101} C_DIS
LIN {X -122.7403,Y -61.8807,Z 176,A -150.9371,B 7.0819,C 0.3288,E1 6.9464,E2 243} C_DIS
LIN {X -124.2432,Y -58.8048,Z 176,A -152.3923,B 7.0821,C 0.3255,E1 6.9446,E2 244.4579} C_DIS
LIN {X -125.6901,Y -55.6455,Z 176,A -153.8531,B 7.0822,C 0.322,E1 6.9429,E2 245.9195} C_DIS
LIN {X -127.0289,Y -52.5171,Z 176,A -155.3109,B 7.0824,C 0.3188,E1 6.9414,E2 247.3813} C_DIS
LIN {X -128.2949,Y -49.3439,Z 176,A -156.7846,B 7.0825,C 0.3156,E1 6.9399,E2 248.8604} C_DIS
LIN {X -129.4738,Y -46.1618,Z 176,A -158.2014,B 7.0827,C 0.3119,E1 6.9385,E2 250.2765} C_DIS
LIN {X -130.5315,Y -43.0794,Z 176,A -159.606,B 7.0828,C 0.3088,E1 6.9372,E2 251.6861} C_DIS
LIN {X -131.6833,Y -39.4257,Z 176,A -161.212,B 7.083,C 0.3046,E1 6.9359,E2 253.2923} C_DIS
LIN {X -132.5059,Y -36.5593,Z 176,A -162.4779,B 7.0831,C 0.3014,E1 6.935,E2 254.5601} C_DIS
LIN {X -133.4355,Y -33.0127,Z 176,A -164.0353,B 7.0833,C 0.2976,E1 6.9339,E2 256.1202} C_DIS
LIN {X -134.1525,Y -29.9625,Z 176,A -165.3585,B 7.0834,C 0.2941,E1 6.9331,E2 257.4445} C_DIS
LIN {X -134.8572,Y -26.6157,Z 176,A -166.8178,B 7.0836,C 0.2906,E1 6.9322,E2 258.9071} C_DIS
LIN {X -135.3688,Y -23.867,Z 176,A -168.0056,B 7.0837,C 0.2876,E1 6.9316,E2 260.0967} C_DIS
LIN {X -135.8876,Y -20.7099,Z 176,A -169.3799,B 7.0838,C 0.2843,E1 6.931,E2 261.475} C_DIS
LIN {X -136.3506,Y -17.4061,Z 176,A -170.7829,B 7.084,C 0.2805,E1 6.9305,E2 262.8785} C_DIS
LIN {X -136.7161,Y -14.2534,Z 176,A -172.1211,B 7.0841,C 0.2769,E1 6.9301,E2 264.2176} C_DIS
LIN {X -136.9621,Y -11.6466,Z 176,A -173.278,B 7.0842,C 0.2746,E1 6.9298,E2 265.3817} C_DIS
LIN {X -137.2239,Y -8.0047,Z 176,A -174.8162,B 7.0844,C 0.2705,E1 6.9295,E2 266.9208} C_DIS
LIN {X -137.3693,Y -4.9131,Z 176,A -176.1308,B 7.0845,C 0.2671,E1 6.9294,E2 268.2374} C_DIS
LIN {X -137.4448,Y -1.8462,Z 176,A -177.3943,B 7.0846,C 0.2632,E1 6.9294,E2 269.498} C_DIS
LIN {X -137.4332,Y 2.5427,Z 176,A -179.2935,B 7.0848,C 0.2588,E1 6.9294,E2 271.4043} C_DIS
LIN {X -137.3405,Y 5.6519,Z 176,A 179.3735,B 7.0849,C 0.2555,E1 6.9294,E2 272.7407} C_DIS
LIN {X -137.1485,Y 9.2287,Z 176,A 177.8628,B 7.0851,C 0.2515,E1 6.9297,E2 274.2523} C_DIS
LIN {X -136.9306,Y 12.0198,Z 176,A 176.6465,B 7.0851,C 0.2487,E1 6.93,E2 275.4737} C_DIS
LIN {X -136.4478,Y 16.6241,Z 176,A 174.6804,B 7.0853,C 0.2437,E1 6.9306,E2 277.4426} C_DIS
LIN {X -136.0336,Y 19.7275,Z 176,A 173.3463,B 7.0855,C 0.2403,E1 6.9311,E2 278.7791} C_DIS
LIN {X -135.5054,Y 23.0807,Z 176,A 171.9125,B 7.0855,C 0.2365,E1 6.9318,E2 280.214} C_DIS
LIN {X -134.8586,Y 26.6091,Z 176,A 170.3837,B 7.0857,C 0.2327,E1 6.9326,E2 281.7457} C_DIS
LIN {X -134.3074,Y 29.2537,Z 176,A 169.2068,B 7.0857,C 0.2301,E1 6.9333,E2 282.9278} C_DIS
LIN {X -133.5174,Y 32.673,Z 176,A 167.7372,B 7.0859,C 0.2261,E1 6.9342,E2 284.3969} C_DIS
LIN {X -132.601,Y 36.2195,Z 176,A 166.177,B 7.086,C 0.2223,E1 6.9353,E2 285.9598} C_DIS
LIN {X -131.6833,Y 39.4257,Z 176,A 164.7563,B 7.0861,C 0.2188,E1 6.9365,E2 287.3831} C_DIS
LIN {X -130.8484,Y 42.1064,Z 176,A 163.539,B 7.0862,C 0.2162,E1 6.9375,E2 288.605} C_DIS
LIN {X -129.5957,Y 45.8239,Z 176,A 161.8907,B 7.0864,C 0.2119,E1 6.939,E2 290.2534} C_DIS
LIN {X -128.5511,Y 48.6724,Z 176,A 160.5987,B 7.0864,C 0.2088,E1 6.9403,E2 291.5476} C_DIS
LIN {X -127.3568,Y 51.7156,Z 176,A 159.1642,B 7.0865,C 0.206,E1 6.9417,E2 292.9896} C_DIS
LIN {X -125.8275,Y 55.3382,Z 176,A 157.5351,B 7.0867,C 0.2016,E1 6.9435,E2 294.616} C_DIS
LIN {X -124.4011,Y 58.4743,Z 176,A 156.0699,B 7.0867,C 0.1982,E1 6.9453,E2 296.0834} C_DIS
LIN {X -122.8897,Y 61.5873,Z 176,A 154.5986,B 7.0868,C 0.1948,E1 6.9471,E2 297.5568} C_DIS
LIN {X -121.2938,Y 64.6737,Z 176,A 153.0743,B 7.0869,C 0.192,E1 6.9491,E2 299.0892} C_DIS
LIN {X -119.2727,Y 68.3284,Z 176,A 151.3471,B 7.087,C 0.1875,E1 6.9514,E2 300.813} C_DIS
LIN {X -117.3972,Y 71.5037,Z 176,A 149.781,B 7.0871,C 0.184,E1 6.9537,E2 302.3813} C_DIS
LIN {X -115.4298,Y 74.6371,Z 176,A 148.1142,B 7.0871,C 0.1819,E1 6.9562,E2 304.0619} C_DIS
LIN {X -112.9787,Y 78.2979,Z 176,A 146.2443,B 7.0873,C 0.1779,E1 6.9591,E2 305.9341} C_DIS
LIN {X -110.6269,Y 81.5869,Z 176,A 144.6025,B 7.0873,C 0.1734,E1 6.9618,E2 307.569} C_DIS
LIN {X -108.2571,Y 84.7062,Z 176,A 142.8678,B 7.0875,C 0.171,E1 6.9648,E2 309.3146} C_DIS
LIN {X -105.7087,Y 87.8659,Z 176,A 141.2441,B 7.0875,C 0.1663,E1 6.9677,E2 310.9284} C_DIS
LIN {X -103.154,Y 90.8515,Z 176,A 139.4829,B 7.0876,C 0.1643,E1 6.9709,E2 312.7031} C_DIS
LIN {X -100.4201,Y 93.8646,Z 176,A 137.7756,B 7.0876,C 0.1609,E1 6.9741,E2 314.4103} C_DIS
LIN {X -97.3308,Y 97.0642,Z 176,A 135.9522,B 7.0878,C 0.1567,E1 6.9777,E2 316.2284} C_DIS
LIN {X -94.6495,Y 99.6812,Z 176,A 134.3421,B 7.0878,C 0.1542,E1 6.9809,E2 317.8429} C_DIS
LIN {X -91.5167,Y 102.5643,Z 176,A 132.5198,B 7.0879,C 0.1514,E1 6.9847,E2 319.6695} C_DIS
LIN {X -88.1549,Y 105.4678,Z 176,A 130.6434,B 7.0879,C 0.1482,E1 6.9887,E2 321.5472} C_DIS
LIN {X -84.7062,Y 108.2571,Z 176,A 128.8416,B 7.088,C 0.1443,E1 6.9926,E2 323.3417} C_DIS
LIN {X -81.738,Y 110.5159,Z 176,A 127.2679,B 7.088,C 0.1419,E1 6.9961,E2 324.9164} C_DIS
LIN {X -78.8688,Y 112.5814,Z 176,A 125.698,B 7.0881,C 0.1407,E1 6.9997,E2 326.4968} C_DIS
LIN {X -75.2187,Y 115.0523,Z 176,A 123.8173,B 7.0881,C 0.1384,E1 7.0041,E2 328.3813} C_DIS
LIN {X -71.5037,Y 117.3972,Z 176,A 122.0687,B 7.0882,C 0.1345,E1 7.0082,E2 330.1182} C_DIS
LIN {X -68.4893,Y 119.1809,Z 176,A 120.5944,B 7.0882,C 0.1326,E1 7.0118,E2 331.5931} C_DIS
LIN {X -65.2782,Y 120.969,Z 176,A 118.9295,B 7.0882,C 0.1322,E1 7.0159,E2 333.273} C_DIS
LIN {X -61.5873,Y 122.8897,Z 176,A 117.2989,B 7.0883,C 0.1286,E1 7.0199,E2 334.8896} C_DIS
LIN {X -58.8048,Y 124.2432,Z 176,A 115.9989,B 7.0883,C 0.1271,E1 7.0232,E2 336.1898} C_DIS
LIN {X -55.8128,Y 125.6152,Z 176,A 114.6003,B 7.0883,C 0.1258,E1 7.0268,E2 337.5907} C_DIS
LIN {X -52.5171,Y 127.0289,Z 176,A 113.1112,B 7.0884,C 0.1241,E1 7.0306,E2 339.078} C_DIS
LIN {X -49.0097,Y 128.4248,Z 176,A 111.5273,B 7.0884,C 0.1226,E1 7.0347,E2 340.6621} C_DIS
LIN {X -46.1618,Y 129.4738,Z 176,A 110.2553,B 7.0884,C 0.1215,E1 7.0381,E2 341.934} C_DIS
LIN {X -43.1298,Y 130.5147,Z 176,A 108.8829,B 7.0884,C 0.1208,E1 7.0417,E2 343.3099} C_DIS
LIN {X -39.8363,Y 131.5576,Z 176,A 107.4581,B 7.0885,C 0.1193,E1 7.0455,E2 344.7319} C_DIS
LIN {X -36.5593,Y 132.5059,Z 176,A 106.037,B 7.0885,C 0.1182,E1 7.0493,E2 346.1519} C_DIS
LIN {X -33.5152,Y 133.308,Z 176,A 104.6975,B 7.0885,C 0.1177,E1 7.053,E2 347.4939} C_DIS
LIN {X -29.8083,Y 134.1877,Z 176,A 103.1263,B 7.0885,C 0.1164,E1 7.0572,E2 349.0621} C_DIS
LIN {X -26.6091,Y 134.8586,Z 176,A 101.7604,B 7.0885,C 0.1157,E1 7.061,E2 350.4276} C_DIS
LIN {X -23.418,Y 135.4491,Z 176,A 100.4052,B 7.0885,C 0.1151,E1 7.0647,E2 351.7824} C_DIS
LIN {X -20.2378,Y 135.9607,Z 176,A 99.0601,B 7.0885,C 0.1145,E1 7.0684,E2 353.1269} C_DIS
LIN {X -17.4061,Y 136.3506,Z 176,A 97.8681,B 7.0885,C 0.1141,E1 7.0717,E2 354.3183} C_DIS
LIN {X -14.2534,Y 136.7161,Z 176,A 96.5445,B 7.0886,C 0.1137,E1 7.0754,E2 355.6413} C_DIS
LIN {X -11.4582,Y 136.978,Z 176,A 95.3301,B 7.0886,C 0.114,E1 7.0788,E2 356.8605} C_DIS
LIN {X -8.0047,Y 137.2239,Z 176,A 93.911,B 7.0886,C 0.1134,E1 7.0827,E2 358.2759} C_DIS
LIN {X -3.7282,Y 137.4059,Z 176,A 92.1035,B 7.0886,C 0.1136,E1 7.0878,E2 360.0853} C_DIS
LIN {X 0,Y 137.4586,Z 176,A 90.5971,B 7.0886,C 0.1129,E1 7.0919,E2 361.5854} C_DIS
LIN {X 3.051,Y 137.4248,Z 176,A 89.323,B 7.0886,C 0.1129,E1 7.0955,E2 362.8591} C_DIS
LIN {X 6.1279,Y 137.322,Z 176,A 88.0384,B 7.0886,C 0.1131,E1 7.0991,E2 364.1434} C_DIS
LIN {X 8.949,Y 137.1657,Z 176,A 86.8481,B 7.0886,C 0.1135,E1 7.1024,E2 365.3347} C_DIS
LIN {X 12.0198,Y 136.9306,Z 176,A 85.5546,B 7.0886,C 0.114,E1 7.106,E2 366.6289} C_DIS
LIN {X 15.4933,Y 136.5827,Z 176,A 84.122,B 7.0886,C 0.1141,E1 7.11,E2 368.0583} C_DIS
LIN {X 18.6525,Y 136.1872,Z 176,A 82.7963,B 7.0886,C 0.1146,E1 7.1136,E2 369.3834} C_DIS
LIN {X 22.7929,Y 135.5534,Z 176,A 81.0252,B 7.0886,C 0.1158,E1 7.1185,E2 371.1569} C_DIS
LIN {X 26.6091,Y 134.8586,Z 176,A 79.4393,B 7.0886,C 0.1162,E1 7.1229,E2 372.7387} C_DIS
LIN {X 29.5277,Y 134.2483,Z 176,A 78.2041,B 7.0886,C 0.1168,E1 7.1263,E2 373.9726} C_DIS
LIN {X 32.673,Y 133.5174,Z 176,A 76.86,B 7.0886,C 0.1177,E1 7.1299,E2 375.316} C_DIS
LIN {X 36.2195,Y 132.601,Z 176,A 75.3378,B 7.0886,C 0.1187,E1 7.134,E2 376.8374} C_DIS
LIN {X 39.4257,Y 131.6833,Z 176,A 73.9536,B 7.0886,C 0.1198,E1 7.1377,E2 378.2207} C_DIS
LIN {X 42.289,Y 130.7901,Z 176,A 72.719,B 7.0885,C 0.1206,E1 7.141,E2 379.453} C_DIS
LIN {X 45.8239,Y 129.5957,Z 176,A 71.163,B 7.0885,C 0.1221,E1 7.1451,E2 381.0089} C_DIS
LIN {X 48.6724,Y 128.5511,Z 176,A 69.9165,B 7.0885,C 0.1231,E1 7.1484,E2 382.2531} C_DIS
LIN {X 52.1822,Y 127.1688,Z 176,A 68.3438,B 7.0885,C 0.1248,E1 7.1524,E2 383.8257} C_DIS
LIN {X 54.9808,Y 125.982,Z 176,A 67.0832,B 7.0884,C 0.1261,E1 7.1557,E2 385.0853} C_DIS
LIN {X 58.4743,Y 124.4011,Z 176,A 65.4994,B 7.0884,C 0.1278,E1 7.1597,E2 386.6673} C_DIS
LIN {X 61.5873,Y 122.8897,Z 176,A 64.0688,B 7.0884,C 0.1294,E1 7.1633,E2 388.0964} C_DIS
LIN {X 64.1524,Y 121.5676,Z 176,A 62.9485,B 7.0884,C 0.1296,E1 7.166,E2 389.2064} C_DIS
LIN {X 67.5689,Y 119.7046,Z 176,A 61.269,B 7.0883,C 0.1328,E1 7.1701,E2 390.8931} C_DIS
LIN {X 70.594,Y 117.9459,Z 176,A 59.8244,B 7.0883,C 0.1347,E1 7.1736,E2 392.336} C_DIS
LIN {X 73.8971,Y 115.905,Z 176,A 58.1295,B 7.0882,C 0.1385,E1 7.1776,E2 394.0405} C_DIS
LIN {X 77.2622,Y 113.6894,Z 176,A 56.5391,B 7.0882,C 0.1397,E1 7.1813,E2 395.62} C_DIS
LIN {X 80.5607,Y 111.3762,Z 176,A 54.8097,B 7.0881,C 0.1433,E1 7.1853,E2 397.3558} C_DIS
LIN {X 84.132,Y 108.7037,Z 176,A 53.0129,B 7.0881,C 0.1455,E1 7.1892,E2 399.1452} C_DIS
LIN {X 87.4658,Y 106.04,Z 176,A 51.2146,B 7.088,C 0.149,E1 7.1931,E2 400.9463} C_DIS
LIN {X 90.8515,Y 103.154,Z 176,A 49.3836,B 7.0879,C 0.1521,E1 7.197,E2 402.7747} C_DIS
LIN {X 93.8646,Y 100.4201,Z 176,A 47.8042,B 7.0879,C 0.1533,E1 7.2002,E2 404.3401} C_DIS
LIN {X 96.5668,Y 97.825,Z 176,A 46.1577,B 7.0878,C 0.1579,E1 7.2035,E2 405.9975} C_DIS
LIN {X 99.6812,Y 94.6495,Z 176,A 44.4377,B 7.0878,C 0.1594,E1 7.2068,E2 407.7015} C_DIS
LIN {X 102.0803,Y 92.0568,Z 176,A 42.9053,B 7.0876,C 0.1636,E1 7.2097,E2 409.2418} C_DIS
LIN {X 105.018,Y 88.691,Z 176,A 41.1544,B 7.0876,C 0.1657,E1 7.2129,E2 410.9795} C_DIS
LIN {X 107.2734,Y 85.9494,Z 176,A 39.6519,B 7.0875,C 0.1693,E1 7.2156,E2 412.4854} C_DIS
LIN {X 109.8463,Y 82.6348,Z 176,A 37.9031,B 7.0875,C 0.1733,E1 7.2185,E2 414.2348} C_DIS
LIN {X 112.4736,Y 79.0218,Z 176,A 36.0793,B 7.0873,C 0.177,E1 7.2215,E2 416.0547} C_DIS
LIN {X 115.0048,Y 75.2907,Z 176,A 34.2265,B 7.0873,C 0.1809,E1 7.2244,E2 417.905} C_DIS
LIN {X 117.3972,Y 71.5037,Z 176,A 32.4666,B 7.0871,C 0.1836,E1 7.2269,E2 419.6525} C_DIS
LIN {X 119.1809,Y 68.4893,Z 176,A 31.0331,B 7.0871,C 0.1867,E1 7.2289,E2 421.0834} C_DIS
LIN {X 120.9647,Y 65.2863,Z 176,A 29.4296,B 7.0869,C 0.1919,E1 7.2311,E2 422.697} C_DIS
LIN {X 122.8897,Y 61.5873,Z 176,A 27.8279,B 7.0869,C 0.1938,E1 7.2331,E2 424.2827} C_DIS
LIN {X 124.1625,Y 58.9737,Z 176,A 26.6199,B 7.0868,C 0.1969,E1 7.2346,E2 425.4908} C_DIS
LIN {X 125.8275,Y 55.3382,Z 176,A 25.0047,B 7.0867,C 0.2003,E1 7.2364,E2 427.1006} C_DIS
LIN {X 127.0289,Y 52.5171,Z 176,A 23.7521,B 7.0867,C 0.2032,E1 7.2378,E2 428.3507} C_DIS
LIN {X 128.4248,Y 49.0097,Z 176,A 22.2097,B 7.0865,C 0.2068,E1 7.2393,E2 429.8903} C_DIS
LIN {X 129.4738,Y 46.1618,Z 176,A 20.9719,B 7.0865,C 0.2097,E1 7.2405,E2 431.1255} C_DIS
LIN {X 130.6817,Y 42.6282,Z 176,A 19.4452,B 7.0863,C 0.2134,E1 7.2419,E2 432.6495} C_DIS
LIN {X 131.6377,Y 39.5748,Z 176,A 18.1497,B 7.0863,C 0.2163,E1 7.2429,E2 433.9411} C_DIS
LIN {X 132.5059,Y 36.5593,Z 176,A 16.8589,B 7.0861,C 0.2196,E1 7.2439,E2 435.2306} C_DIS
LIN {X 133.4355,Y 33.0127,Z 176,A 15.3624,B 7.0861,C 0.2233,E1 7.2449,E2 436.7242} C_DIS
LIN {X 134.1877,Y 29.8083,Z 176,A 14.0192,B 7.0859,C 0.2266,E1 7.2458,E2 438.0648} C_DIS
LIN {X 134.8015,Y 26.8895,Z 176,A 12.8159,B 7.0859,C 0.2293,E1 7.2465,E2 439.2639} C_DIS
LIN {X 135.3534,Y 23.953,Z 176,A 11.5348,B 7.0857,C 0.2335,E1 7.2471,E2 440.5504} C_DIS
LIN {X 135.9607,Y 20.2378,Z 176,A 10.0482,B 7.0856,C 0.2364,E1 7.2477,E2 442.028} C_DIS
LIN {X 136.3506,Y 17.4061,Z 176,A 8.8831,B 7.0855,C 0.2393,E1 7.2482,E2 443.1905} C_DIS
LIN {X 136.7161,Y 14.2534,Z 176,A 7.589,B 7.0854,C 0.2426,E1 7.2486,E2 444.4821} C_DIS
Enddeposition()
END
